REGION Network 4: 3号梯内呼指示灯绑定
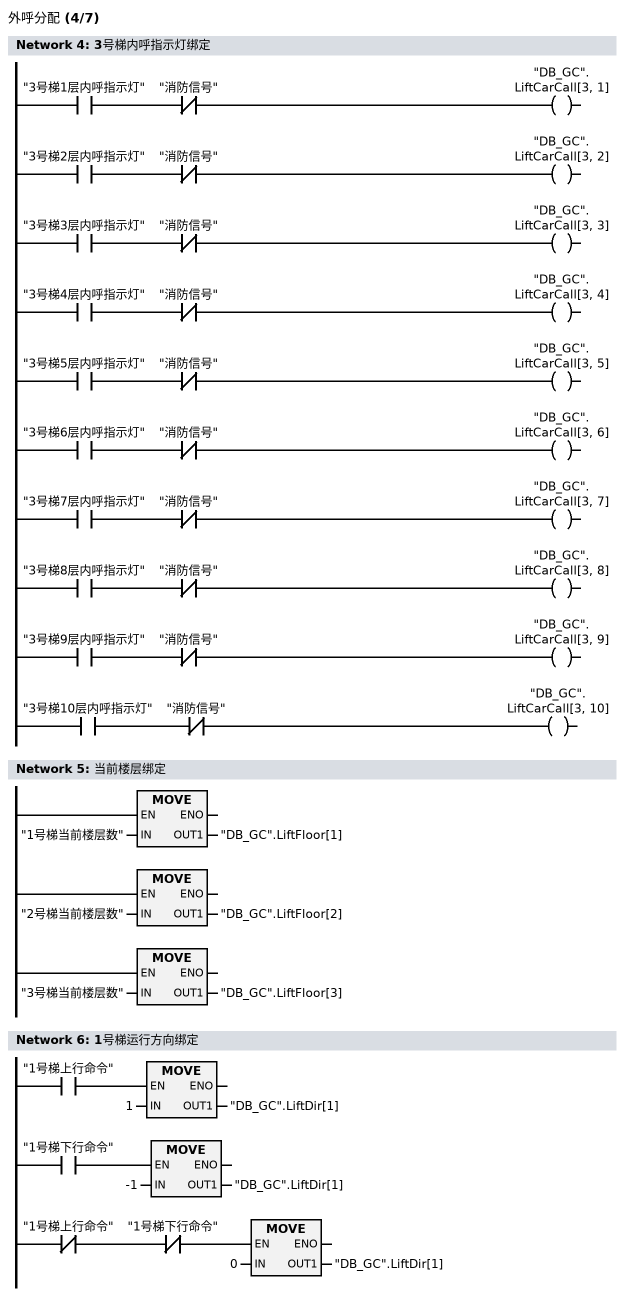
   RUNG wire#powerrail
      Contact( "3号梯1层内呼指示灯" )
      I_Contact( "消防信号" )
      Coil( "DB_GC".LiftCarCall[3, 1] )
   END_RUNG
   RUNG wire#powerrail
      Contact( "3号梯2层内呼指示灯" )
      I_Contact( "消防信号" )
      Coil( "DB_GC".LiftCarCall[3, 2] )
   END_RUNG
   RUNG wire#powerrail
      Contact( "3号梯3层内呼指示灯" )
      I_Contact( "消防信号" )
      Coil( "DB_GC".LiftCarCall[3, 3] )
   END_RUNG
   RUNG wire#powerrail
      Contact( "3号梯4层内呼指示灯" )
      I_Contact( "消防信号" )
      Coil( "DB_GC".LiftCarCall[3, 4] )
   END_RUNG
   RUNG wire#powerrail
      Contact( "3号梯5层内呼指示灯" )
      I_Contact( "消防信号" )
      Coil( "DB_GC".LiftCarCall[3, 5] )
   END_RUNG
   RUNG wire#powerrail
      Contact( "3号梯6层内呼指示灯" )
      I_Contact( "消防信号" )
      Coil( "DB_GC".LiftCarCall[3, 6] )
   END_RUNG
   RUNG wire#powerrail
      Contact( "3号梯7层内呼指示灯" )
      I_Contact( "消防信号" )
      Coil( "DB_GC".LiftCarCall[3, 7] )
   END_RUNG
   RUNG wire#powerrail
      Contact( "3号梯8层内呼指示灯" )
      I_Contact( "消防信号" )
      Coil( "DB_GC".LiftCarCall[3, 8] )
   END_RUNG
   RUNG wire#powerrail
      Contact( "3号梯9层内呼指示灯" )
      I_Contact( "消防信号" )
      Coil( "DB_GC".LiftCarCall[3, 9] )
   END_RUNG
   RUNG wire#powerrail
      Contact( "3号梯10层内呼指示灯" )
      I_Contact( "消防信号" )
      Coil( "DB_GC".LiftCarCall[3, 10] )
   END_RUNG
   // the same network as SCL:
   "DB_GC".LiftCarCall[3, 1] := "3号梯1层内呼指示灯" AND NOT "消防信号";
   "DB_GC".LiftCarCall[3, 2] := "3号梯2层内呼指示灯" AND NOT "消防信号";
   "DB_GC".LiftCarCall[3, 3] := "3号梯3层内呼指示灯" AND NOT "消防信号";
   "DB_GC".LiftCarCall[3, 4] := "3号梯4层内呼指示灯" AND NOT "消防信号";
   "DB_GC".LiftCarCall[3, 5] := "3号梯5层内呼指示灯" AND NOT "消防信号";
   "DB_GC".LiftCarCall[3, 6] := "3号梯6层内呼指示灯" AND NOT "消防信号";
   "DB_GC".LiftCarCall[3, 7] := "3号梯7层内呼指示灯" AND NOT "消防信号";
   "DB_GC".LiftCarCall[3, 8] := "3号梯8层内呼指示灯" AND NOT "消防信号";
   "DB_GC".LiftCarCall[3, 9] := "3号梯9层内呼指示灯" AND NOT "消防信号";
   "DB_GC".LiftCarCall[3, 10] := "3号梯10层内呼指示灯" AND NOT "消防信号";
END_REGION

REGION Network 5: 当前楼层绑定
   RUNG wire#powerrail
      Move(in := "1号梯当前楼层数", out1 => "DB_GC".LiftFloor[1])
   END_RUNG
   RUNG wire#powerrail
      Move(in := "2号梯当前楼层数", out1 => "DB_GC".LiftFloor[2])
   END_RUNG
   RUNG wire#powerrail
      Move(in := "3号梯当前楼层数", out1 => "DB_GC".LiftFloor[3])
   END_RUNG
   // the same network as SCL:
   "DB_GC".LiftFloor[1] := "1号梯当前楼层数";
   "DB_GC".LiftFloor[2] := "2号梯当前楼层数";
   "DB_GC".LiftFloor[3] := "3号梯当前楼层数";
END_REGION

REGION Network 6: 1号梯运行方向绑定
   RUNG wire#powerrail
      Contact( "1号梯上行命令" )
      Move(in := 1, out1 => "DB_GC".LiftDir[1])
   END_RUNG
   RUNG wire#powerrail
      Contact( "1号梯下行命令" )
      Move(in := -1, out1 => "DB_GC".LiftDir[1])
   END_RUNG
   RUNG wire#powerrail
      I_Contact( "1号梯上行命令" )
      I_Contact( "1号梯下行命令" )
      Move(in := 0, out1 => "DB_GC".LiftDir[1])
   END_RUNG
   // the same network as SCL:
   IF "1号梯上行命令" THEN "DB_GC".LiftDir[1] := 1; END_IF;
   IF "1号梯下行命令" THEN "DB_GC".LiftDir[1] := -1; END_IF;
   IF NOT "1号梯上行命令" AND NOT "1号梯下行命令" THEN "DB_GC".LiftDir[1] := 0; END_IF;
END_REGION

REGION Network 7: 2号梯运行方向绑定
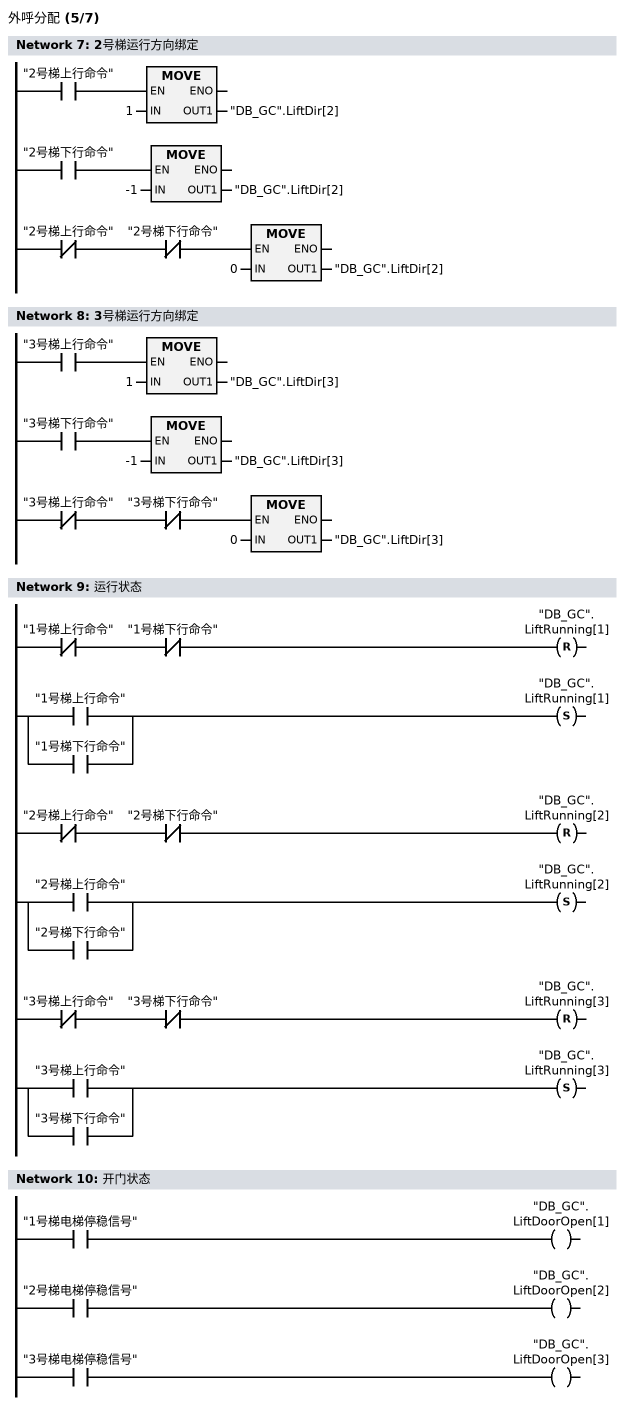
   RUNG wire#powerrail
      Contact( "2号梯上行命令" )
      Move(in := 1, out1 => "DB_GC".LiftDir[2])
   END_RUNG
   RUNG wire#powerrail
      Contact( "2号梯下行命令" )
      Move(in := -1, out1 => "DB_GC".LiftDir[2])
   END_RUNG
   RUNG wire#powerrail
      I_Contact( "2号梯上行命令" )
      I_Contact( "2号梯下行命令" )
      Move(in := 0, out1 => "DB_GC".LiftDir[2])
   END_RUNG
   // the same network as SCL:
   IF "2号梯上行命令" THEN "DB_GC".LiftDir[2] := 1; END_IF;
   IF "2号梯下行命令" THEN "DB_GC".LiftDir[2] := -1; END_IF;
   IF NOT "2号梯上行命令" AND NOT "2号梯下行命令" THEN "DB_GC".LiftDir[2] := 0; END_IF;
END_REGION

REGION Network 8: 3号梯运行方向绑定
   RUNG wire#powerrail
      Contact( "3号梯上行命令" )
      Move(in := 1, out1 => "DB_GC".LiftDir[3])
   END_RUNG
   RUNG wire#powerrail
      Contact( "3号梯下行命令" )
      Move(in := -1, out1 => "DB_GC".LiftDir[3])
   END_RUNG
   RUNG wire#powerrail
      I_Contact( "3号梯上行命令" )
      I_Contact( "3号梯下行命令" )
      Move(in := 0, out1 => "DB_GC".LiftDir[3])
   END_RUNG
   // the same network as SCL:
   IF "3号梯上行命令" THEN "DB_GC".LiftDir[3] := 1; END_IF;
   IF "3号梯下行命令" THEN "DB_GC".LiftDir[3] := -1; END_IF;
   IF NOT "3号梯上行命令" AND NOT "3号梯下行命令" THEN "DB_GC".LiftDir[3] := 0; END_IF;
END_REGION

REGION Network 9: 运行状态
   RUNG wire#powerrail
      I_Contact( "1号梯上行命令" )
      I_Contact( "1号梯下行命令" )
      R_Coil( "DB_GC".LiftRunning[1] )
   END_RUNG
   RUNG wire#powerrail
      Contact( "1号梯上行命令" )
      wire#w1
      S_Coil( "DB_GC".LiftRunning[1] )
   END_RUNG
   RUNG wire#powerrail
      Contact( "1号梯下行命令" )
   END_RUNG wire#w1
   RUNG wire#powerrail
      I_Contact( "2号梯上行命令" )
      I_Contact( "2号梯下行命令" )
      R_Coil( "DB_GC".LiftRunning[2] )
   END_RUNG
   RUNG wire#powerrail
      Contact( "2号梯上行命令" )
      wire#w2
      S_Coil( "DB_GC".LiftRunning[2] )
   END_RUNG
   RUNG wire#powerrail
      Contact( "2号梯下行命令" )
   END_RUNG wire#w2
   RUNG wire#powerrail
      I_Contact( "3号梯上行命令" )
      I_Contact( "3号梯下行命令" )
      R_Coil( "DB_GC".LiftRunning[3] )
   END_RUNG
   RUNG wire#powerrail
      Contact( "3号梯上行命令" )
      wire#w3
      S_Coil( "DB_GC".LiftRunning[3] )
   END_RUNG
   RUNG wire#powerrail
      Contact( "3号梯下行命令" )
   END_RUNG wire#w3
   // the same network as SCL:
   IF NOT "1号梯上行命令" AND NOT "1号梯下行命令" THEN "DB_GC".LiftRunning[1] := FALSE; END_IF;
   IF "1号梯上行命令" OR "1号梯下行命令" THEN "DB_GC".LiftRunning[1] := TRUE; END_IF;
   IF NOT "2号梯上行命令" AND NOT "2号梯下行命令" THEN "DB_GC".LiftRunning[2] := FALSE; END_IF;
   IF "2号梯上行命令" OR "2号梯下行命令" THEN "DB_GC".LiftRunning[2] := TRUE; END_IF;
   IF NOT "3号梯上行命令" AND NOT "3号梯下行命令" THEN "DB_GC".LiftRunning[3] := FALSE; END_IF;
   IF "3号梯上行命令" OR "3号梯下行命令" THEN "DB_GC".LiftRunning[3] := TRUE; END_IF;
END_REGION

REGION Network 10: 开门状态
   RUNG wire#powerrail
      Contact( "1号梯电梯停稳信号" )
      Coil( "DB_GC".LiftDoorOpen[1] )
   END_RUNG
   RUNG wire#powerrail
      Contact( "2号梯电梯停稳信号" )
      Coil( "DB_GC".LiftDoorOpen[2] )
   END_RUNG
   RUNG wire#powerrail
      Contact( "3号梯电梯停稳信号" )
      Coil( "DB_GC".LiftDoorOpen[3] )
   END_RUNG
   // the same network as SCL:
   "DB_GC".LiftDoorOpen[1] := "1号梯电梯停稳信号";
   "DB_GC".LiftDoorOpen[2] := "2号梯电梯停稳信号";
   "DB_GC".LiftDoorOpen[3] := "3号梯电梯停稳信号";
END_REGION

REGION Network 11: 锁梯
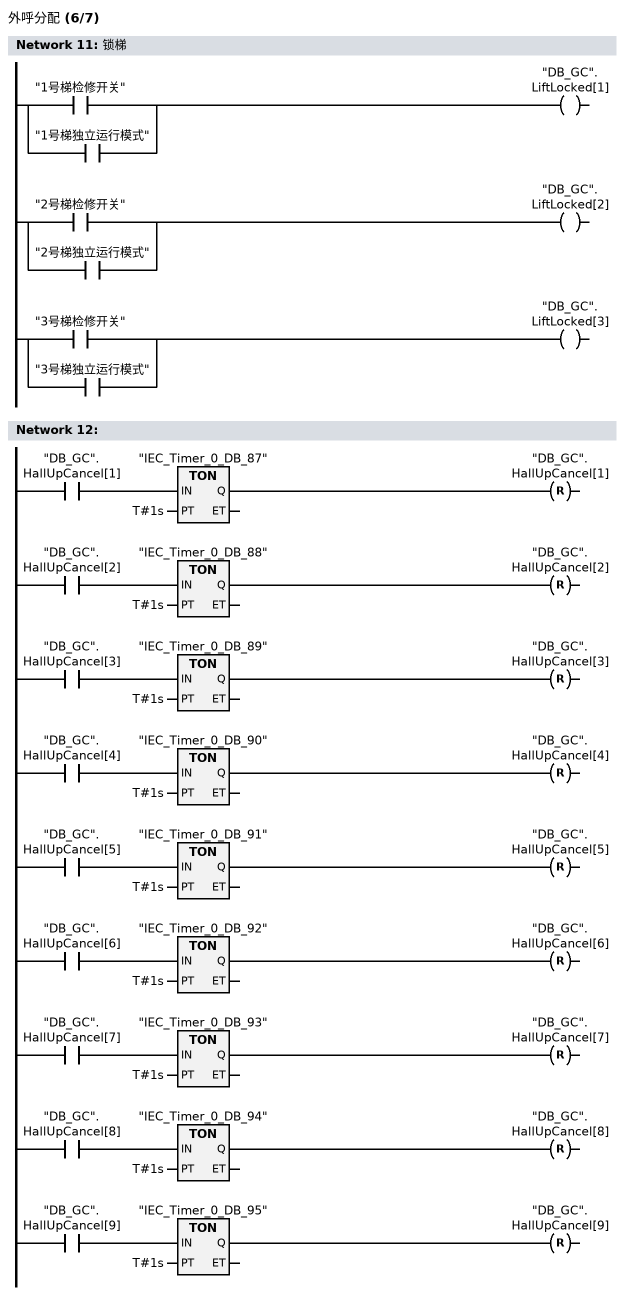
   RUNG wire#powerrail
      Contact( "1号梯检修开关" )
      wire#w1
      Coil( "DB_GC".LiftLocked[1] )
   END_RUNG
   RUNG wire#powerrail
      Contact( "1号梯独立运行模式" )
   END_RUNG wire#w1
   RUNG wire#powerrail
      Contact( "2号梯检修开关" )
      wire#w2
      Coil( "DB_GC".LiftLocked[2] )
   END_RUNG
   RUNG wire#powerrail
      Contact( "2号梯独立运行模式" )
   END_RUNG wire#w2
   RUNG wire#powerrail
      Contact( "3号梯检修开关" )
      wire#w3
      Coil( "DB_GC".LiftLocked[3] )
   END_RUNG
   RUNG wire#powerrail
      Contact( "3号梯独立运行模式" )
   END_RUNG wire#w3
   // the same network as SCL:
   "DB_GC".LiftLocked[1] := "1号梯检修开关" OR "1号梯独立运行模式";
   "DB_GC".LiftLocked[2] := "2号梯检修开关" OR "2号梯独立运行模式";
   "DB_GC".LiftLocked[3] := "3号梯检修开关" OR "3号梯独立运行模式";
END_REGION

REGION Network 12
   "IEC_Timer_0_DB_87".TON(IN := "DB_GC".HallUpCancel[1], PT := T#1s);
   IF "IEC_Timer_0_DB_87".Q THEN "DB_GC".HallUpCancel[1] := FALSE; END_IF;
   "IEC_Timer_0_DB_88".TON(IN := "DB_GC".HallUpCancel[2], PT := T#1s);
   IF "IEC_Timer_0_DB_88".Q THEN "DB_GC".HallUpCancel[2] := FALSE; END_IF;
   "IEC_Timer_0_DB_89".TON(IN := "DB_GC".HallUpCancel[3], PT := T#1s);
   IF "IEC_Timer_0_DB_89".Q THEN "DB_GC".HallUpCancel[3] := FALSE; END_IF;
   "IEC_Timer_0_DB_90".TON(IN := "DB_GC".HallUpCancel[4], PT := T#1s);
   IF "IEC_Timer_0_DB_90".Q THEN "DB_GC".HallUpCancel[4] := FALSE; END_IF;
   "IEC_Timer_0_DB_91".TON(IN := "DB_GC".HallUpCancel[5], PT := T#1s);
   IF "IEC_Timer_0_DB_91".Q THEN "DB_GC".HallUpCancel[5] := FALSE; END_IF;
   "IEC_Timer_0_DB_92".TON(IN := "DB_GC".HallUpCancel[6], PT := T#1s);
   IF "IEC_Timer_0_DB_92".Q THEN "DB_GC".HallUpCancel[6] := FALSE; END_IF;
   "IEC_Timer_0_DB_93".TON(IN := "DB_GC".HallUpCancel[7], PT := T#1s);
   IF "IEC_Timer_0_DB_93".Q THEN "DB_GC".HallUpCancel[7] := FALSE; END_IF;
   "IEC_Timer_0_DB_94".TON(IN := "DB_GC".HallUpCancel[8], PT := T#1s);
   IF "IEC_Timer_0_DB_94".Q THEN "DB_GC".HallUpCancel[8] := FALSE; END_IF;
   "IEC_Timer_0_DB_95".TON(IN := "DB_GC".HallUpCancel[9], PT := T#1s);
   IF "IEC_Timer_0_DB_95".Q THEN "DB_GC".HallUpCancel[9] := FALSE; END_IF;
END_REGION

REGION Network 13
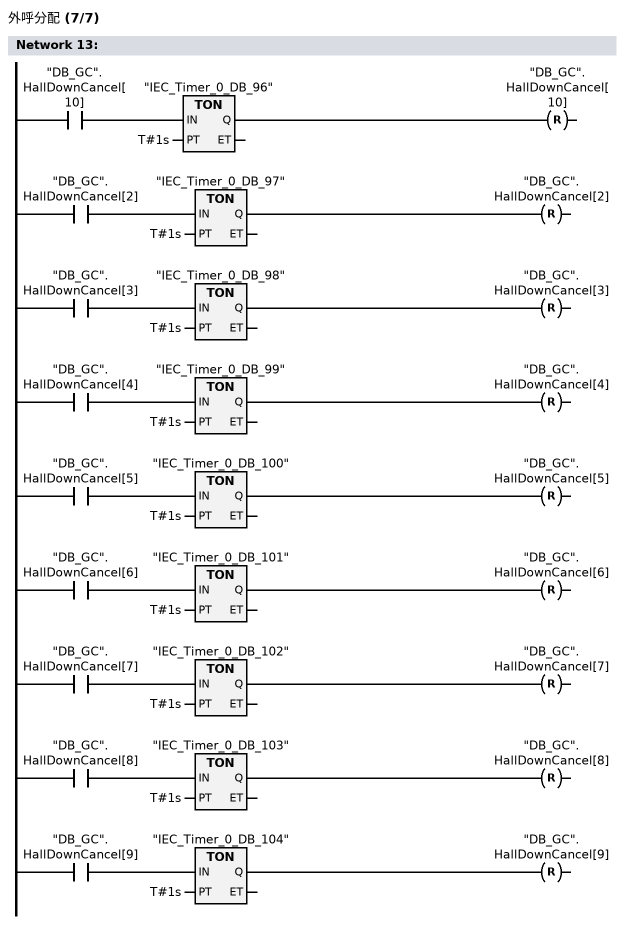
   "IEC_Timer_0_DB_96".TON(IN := "DB_GC".HallDownCancel[10], PT := T#1s);
   IF "IEC_Timer_0_DB_96".Q THEN "DB_GC".HallDownCancel[10] := FALSE; END_IF;
   "IEC_Timer_0_DB_97".TON(IN := "DB_GC".HallDownCancel[2], PT := T#1s);
   IF "IEC_Timer_0_DB_97".Q THEN "DB_GC".HallDownCancel[2] := FALSE; END_IF;
   "IEC_Timer_0_DB_98".TON(IN := "DB_GC".HallDownCancel[3], PT := T#1s);
   IF "IEC_Timer_0_DB_98".Q THEN "DB_GC".HallDownCancel[3] := FALSE; END_IF;
   "IEC_Timer_0_DB_99".TON(IN := "DB_GC".HallDownCancel[4], PT := T#1s);
   IF "IEC_Timer_0_DB_99".Q THEN "DB_GC".HallDownCancel[4] := FALSE; END_IF;
   "IEC_Timer_0_DB_100".TON(IN := "DB_GC".HallDownCancel[5], PT := T#1s);
   IF "IEC_Timer_0_DB_100".Q THEN "DB_GC".HallDownCancel[5] := FALSE; END_IF;
   "IEC_Timer_0_DB_101".TON(IN := "DB_GC".HallDownCancel[6], PT := T#1s);
   IF "IEC_Timer_0_DB_101".Q THEN "DB_GC".HallDownCancel[6] := FALSE; END_IF;
   "IEC_Timer_0_DB_102".TON(IN := "DB_GC".HallDownCancel[7], PT := T#1s);
   IF "IEC_Timer_0_DB_102".Q THEN "DB_GC".HallDownCancel[7] := FALSE; END_IF;
   "IEC_Timer_0_DB_103".TON(IN := "DB_GC".HallDownCancel[8], PT := T#1s);
   IF "IEC_Timer_0_DB_103".Q THEN "DB_GC".HallDownCancel[8] := FALSE; END_IF;
   "IEC_Timer_0_DB_104".TON(IN := "DB_GC".HallDownCancel[9], PT := T#1s);
   IF "IEC_Timer_0_DB_104".Q THEN "DB_GC".HallDownCancel[9] := FALSE; END_IF;
END_REGION
END_FUNCTION

FUNCTION "变量输出赋值" : Void   // FC2, LAD
{ S7_Optimized_Access := 'TRUE' }
VERSION : 0.1
   VAR_TEMP
      沿 : Bool;
   END_VAR
   VAR_TEMP   // added for the SCL form of the ladder/FBD networks
      _w1 : Bool;
   END_VAR
BEGIN

REGION Network 1: 1号梯内呼指示灯
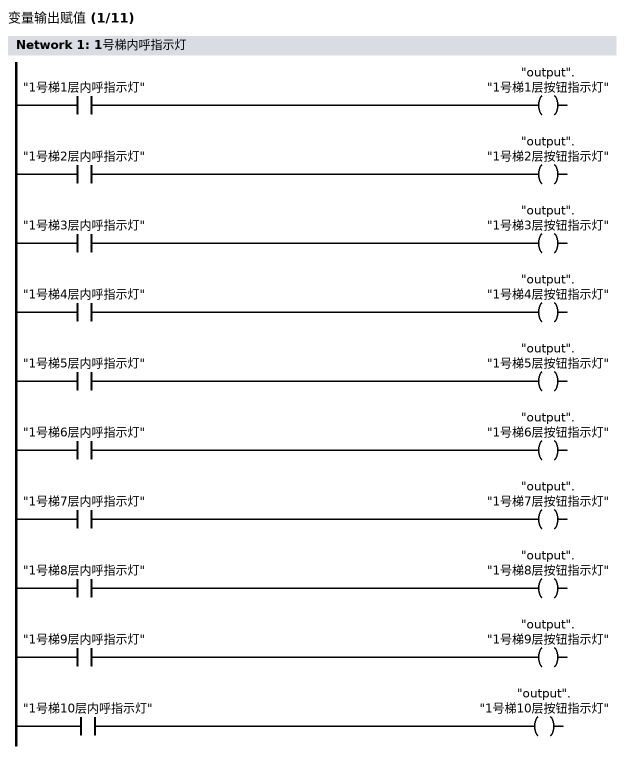
   RUNG wire#powerrail
      Contact( "1号梯1层内呼指示灯" )
      Coil( "output"."1号梯1层按钮指示灯" )
   END_RUNG
   RUNG wire#powerrail
      Contact( "1号梯2层内呼指示灯" )
      Coil( "output"."1号梯2层按钮指示灯" )
   END_RUNG
   RUNG wire#powerrail
      Contact( "1号梯3层内呼指示灯" )
      Coil( "output"."1号梯3层按钮指示灯" )
   END_RUNG
   RUNG wire#powerrail
      Contact( "1号梯4层内呼指示灯" )
      Coil( "output"."1号梯4层按钮指示灯" )
   END_RUNG
   RUNG wire#powerrail
      Contact( "1号梯5层内呼指示灯" )
      Coil( "output"."1号梯5层按钮指示灯" )
   END_RUNG
   RUNG wire#powerrail
      Contact( "1号梯6层内呼指示灯" )
      Coil( "output"."1号梯6层按钮指示灯" )
   END_RUNG
   RUNG wire#powerrail
      Contact( "1号梯7层内呼指示灯" )
      Coil( "output"."1号梯7层按钮指示灯" )
   END_RUNG
   RUNG wire#powerrail
      Contact( "1号梯8层内呼指示灯" )
      Coil( "output"."1号梯8层按钮指示灯" )
   END_RUNG
   RUNG wire#powerrail
      Contact( "1号梯9层内呼指示灯" )
      Coil( "output"."1号梯9层按钮指示灯" )
   END_RUNG
   RUNG wire#powerrail
      Contact( "1号梯10层内呼指示灯" )
      Coil( "output"."1号梯10层按钮指示灯" )
   END_RUNG
   // the same network as SCL:
   "output"."1号梯1层按钮指示灯" := "1号梯1层内呼指示灯";
   "output"."1号梯2层按钮指示灯" := "1号梯2层内呼指示灯";
   "output"."1号梯3层按钮指示灯" := "1号梯3层内呼指示灯";
   "output"."1号梯4层按钮指示灯" := "1号梯4层内呼指示灯";
   "output"."1号梯5层按钮指示灯" := "1号梯5层内呼指示灯";
   "output"."1号梯6层按钮指示灯" := "1号梯6层内呼指示灯";
   "output"."1号梯7层按钮指示灯" := "1号梯7层内呼指示灯";
   "output"."1号梯8层按钮指示灯" := "1号梯8层内呼指示灯";
   "output"."1号梯9层按钮指示灯" := "1号梯9层内呼指示灯";
   "output"."1号梯10层按钮指示灯" := "1号梯10层内呼指示灯";
END_REGION

REGION Network 2: 2号梯内呼指示灯
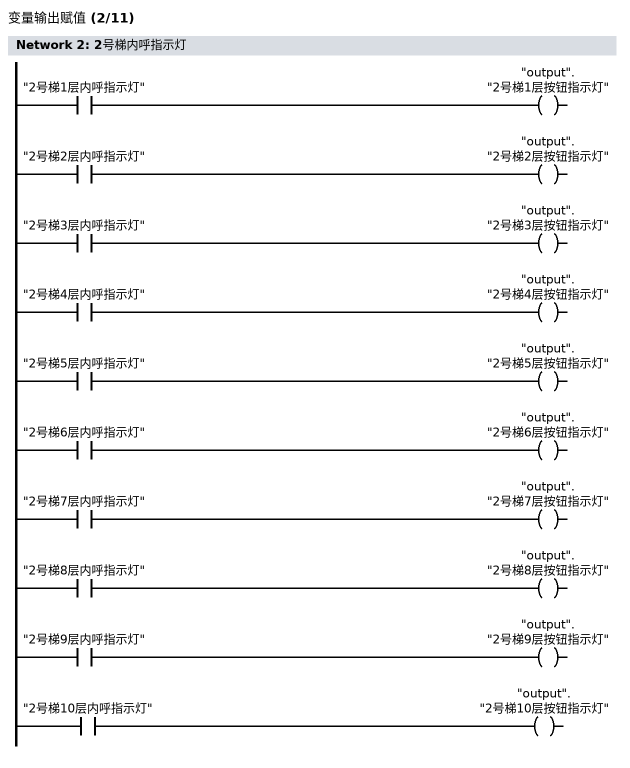
   RUNG wire#powerrail
      Contact( "2号梯1层内呼指示灯" )
      Coil( "output"."2号梯1层按钮指示灯" )
   END_RUNG
   RUNG wire#powerrail
      Contact( "2号梯2层内呼指示灯" )
      Coil( "output"."2号梯2层按钮指示灯" )
   END_RUNG
   RUNG wire#powerrail
      Contact( "2号梯3层内呼指示灯" )
      Coil( "output"."2号梯3层按钮指示灯" )
   END_RUNG
   RUNG wire#powerrail
      Contact( "2号梯4层内呼指示灯" )
      Coil( "output"."2号梯4层按钮指示灯" )
   END_RUNG
   RUNG wire#powerrail
      Contact( "2号梯5层内呼指示灯" )
      Coil( "output"."2号梯5层按钮指示灯" )
   END_RUNG
   RUNG wire#powerrail
      Contact( "2号梯6层内呼指示灯" )
      Coil( "output"."2号梯6层按钮指示灯" )
   END_RUNG
   RUNG wire#powerrail
      Contact( "2号梯7层内呼指示灯" )
      Coil( "output"."2号梯7层按钮指示灯" )
   END_RUNG
   RUNG wire#powerrail
      Contact( "2号梯8层内呼指示灯" )
      Coil( "output"."2号梯8层按钮指示灯" )
   END_RUNG
   RUNG wire#powerrail
      Contact( "2号梯9层内呼指示灯" )
      Coil( "output"."2号梯9层按钮指示灯" )
   END_RUNG
   RUNG wire#powerrail
      Contact( "2号梯10层内呼指示灯" )
      Coil( "output"."2号梯10层按钮指示灯" )
   END_RUNG
   // the same network as SCL:
   "output"."2号梯1层按钮指示灯" := "2号梯1层内呼指示灯";
   "output"."2号梯2层按钮指示灯" := "2号梯2层内呼指示灯";
   "output"."2号梯3层按钮指示灯" := "2号梯3层内呼指示灯";
   "output"."2号梯4层按钮指示灯" := "2号梯4层内呼指示灯";
   "output"."2号梯5层按钮指示灯" := "2号梯5层内呼指示灯";
   "output"."2号梯6层按钮指示灯" := "2号梯6层内呼指示灯";
   "output"."2号梯7层按钮指示灯" := "2号梯7层内呼指示灯";
   "output"."2号梯8层按钮指示灯" := "2号梯8层内呼指示灯";
   "output"."2号梯9层按钮指示灯" := "2号梯9层内呼指示灯";
   "output"."2号梯10层按钮指示灯" := "2号梯10层内呼指示灯";
END_REGION

REGION Network 3: 3号梯内呼指示灯
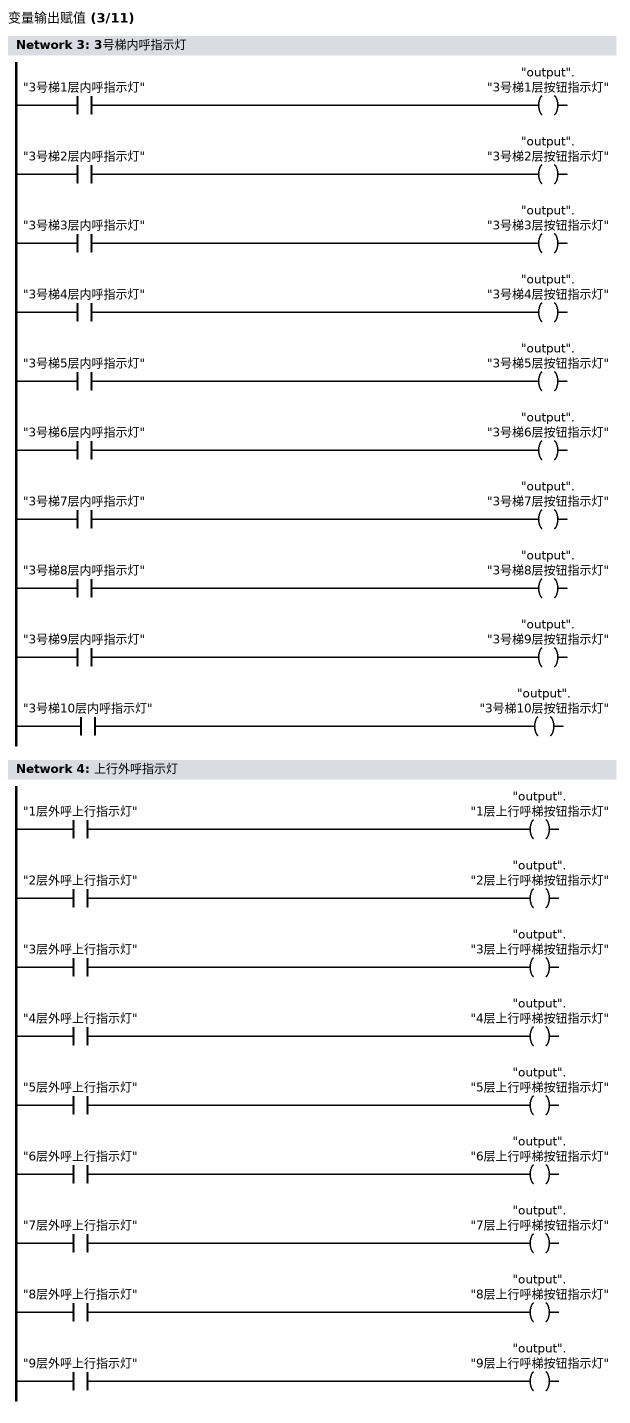
   RUNG wire#powerrail
      Contact( "3号梯1层内呼指示灯" )
      Coil( "output"."3号梯1层按钮指示灯" )
   END_RUNG
   RUNG wire#powerrail
      Contact( "3号梯2层内呼指示灯" )
      Coil( "output"."3号梯2层按钮指示灯" )
   END_RUNG
   RUNG wire#powerrail
      Contact( "3号梯3层内呼指示灯" )
      Coil( "output"."3号梯3层按钮指示灯" )
   END_RUNG
   RUNG wire#powerrail
      Contact( "3号梯4层内呼指示灯" )
      Coil( "output"."3号梯4层按钮指示灯" )
   END_RUNG
   RUNG wire#powerrail
      Contact( "3号梯5层内呼指示灯" )
      Coil( "output"."3号梯5层按钮指示灯" )
   END_RUNG
   RUNG wire#powerrail
      Contact( "3号梯6层内呼指示灯" )
      Coil( "output"."3号梯6层按钮指示灯" )
   END_RUNG
   RUNG wire#powerrail
      Contact( "3号梯7层内呼指示灯" )
      Coil( "output"."3号梯7层按钮指示灯" )
   END_RUNG
   RUNG wire#powerrail
      Contact( "3号梯8层内呼指示灯" )
      Coil( "output"."3号梯8层按钮指示灯" )
   END_RUNG
   RUNG wire#powerrail
      Contact( "3号梯9层内呼指示灯" )
      Coil( "output"."3号梯9层按钮指示灯" )
   END_RUNG
   RUNG wire#powerrail
      Contact( "3号梯10层内呼指示灯" )
      Coil( "output"."3号梯10层按钮指示灯" )
   END_RUNG
   // the same network as SCL:
   "output"."3号梯1层按钮指示灯" := "3号梯1层内呼指示灯";
   "output"."3号梯2层按钮指示灯" := "3号梯2层内呼指示灯";
   "output"."3号梯3层按钮指示灯" := "3号梯3层内呼指示灯";
   "output"."3号梯4层按钮指示灯" := "3号梯4层内呼指示灯";
   "output"."3号梯5层按钮指示灯" := "3号梯5层内呼指示灯";
   "output"."3号梯6层按钮指示灯" := "3号梯6层内呼指示灯";
   "output"."3号梯7层按钮指示灯" := "3号梯7层内呼指示灯";
   "output"."3号梯8层按钮指示灯" := "3号梯8层内呼指示灯";
   "output"."3号梯9层按钮指示灯" := "3号梯9层内呼指示灯";
   "output"."3号梯10层按钮指示灯" := "3号梯10层内呼指示灯";
END_REGION

REGION Network 4: 上行外呼指示灯
   RUNG wire#powerrail
      Contact( "1层外呼上行指示灯" )
      Coil( "output"."1层上行呼梯按钮指示灯" )
   END_RUNG
   RUNG wire#powerrail
      Contact( "2层外呼上行指示灯" )
      Coil( "output"."2层上行呼梯按钮指示灯" )
   END_RUNG
   RUNG wire#powerrail
      Contact( "3层外呼上行指示灯" )
      Coil( "output"."3层上行呼梯按钮指示灯" )
   END_RUNG
   RUNG wire#powerrail
      Contact( "4层外呼上行指示灯" )
      Coil( "output"."4层上行呼梯按钮指示灯" )
   END_RUNG
   RUNG wire#powerrail
      Contact( "5层外呼上行指示灯" )
      Coil( "output"."5层上行呼梯按钮指示灯" )
   END_RUNG
   RUNG wire#powerrail
      Contact( "6层外呼上行指示灯" )
      Coil( "output"."6层上行呼梯按钮指示灯" )
   END_RUNG
   RUNG wire#powerrail
      Contact( "7层外呼上行指示灯" )
      Coil( "output"."7层上行呼梯按钮指示灯" )
   END_RUNG
   RUNG wire#powerrail
      Contact( "8层外呼上行指示灯" )
      Coil( "output"."8层上行呼梯按钮指示灯" )
   END_RUNG
   RUNG wire#powerrail
      Contact( "9层外呼上行指示灯" )
      Coil( "output"."9层上行呼梯按钮指示灯" )
   END_RUNG
   // the same network as SCL:
   "output"."1层上行呼梯按钮指示灯" := "1层外呼上行指示灯";
   "output"."2层上行呼梯按钮指示灯" := "2层外呼上行指示灯";
   "output"."3层上行呼梯按钮指示灯" := "3层外呼上行指示灯";
   "output"."4层上行呼梯按钮指示灯" := "4层外呼上行指示灯";
   "output"."5层上行呼梯按钮指示灯" := "5层外呼上行指示灯";
   "output"."6层上行呼梯按钮指示灯" := "6层外呼上行指示灯";
   "output"."7层上行呼梯按钮指示灯" := "7层外呼上行指示灯";
   "output"."8层上行呼梯按钮指示灯" := "8层外呼上行指示灯";
   "output"."9层上行呼梯按钮指示灯" := "9层外呼上行指示灯";
END_REGION

REGION Network 5: 下行外呼指示灯
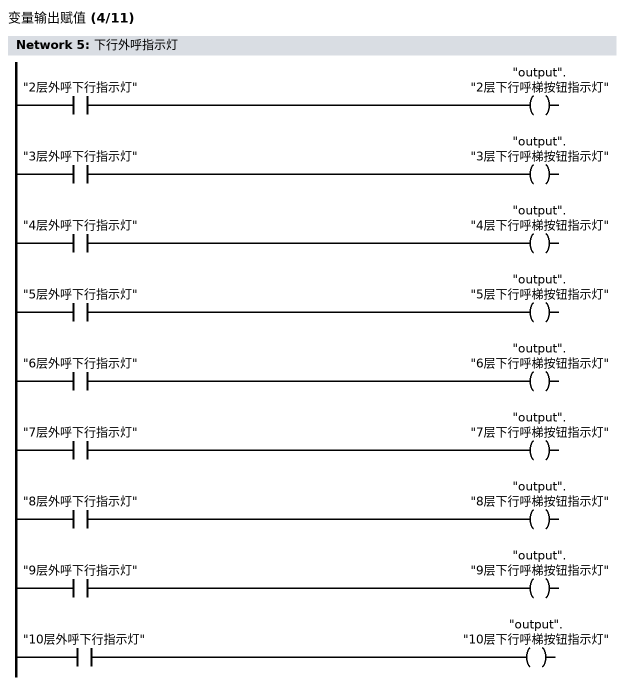
   RUNG wire#powerrail
      Contact( "2层外呼下行指示灯" )
      Coil( "output"."2层下行呼梯按钮指示灯" )
   END_RUNG
   RUNG wire#powerrail
      Contact( "3层外呼下行指示灯" )
      Coil( "output"."3层下行呼梯按钮指示灯" )
   END_RUNG
   RUNG wire#powerrail
      Contact( "4层外呼下行指示灯" )
      Coil( "output"."4层下行呼梯按钮指示灯" )
   END_RUNG
   RUNG wire#powerrail
      Contact( "5层外呼下行指示灯" )
      Coil( "output"."5层下行呼梯按钮指示灯" )
   END_RUNG
   RUNG wire#powerrail
      Contact( "6层外呼下行指示灯" )
      Coil( "output"."6层下行呼梯按钮指示灯" )
   END_RUNG
   RUNG wire#powerrail
      Contact( "7层外呼下行指示灯" )
      Coil( "output"."7层下行呼梯按钮指示灯" )
   END_RUNG
   RUNG wire#powerrail
      Contact( "8层外呼下行指示灯" )
      Coil( "output"."8层下行呼梯按钮指示灯" )
   END_RUNG
   RUNG wire#powerrail
      Contact( "9层外呼下行指示灯" )
      Coil( "output"."9层下行呼梯按钮指示灯" )
   END_RUNG
   RUNG wire#powerrail
      Contact( "10层外呼下行指示灯" )
      Coil( "output"."10层下行呼梯按钮指示灯" )
   END_RUNG
   // the same network as SCL:
   "output"."2层下行呼梯按钮指示灯" := "2层外呼下行指示灯";
   "output"."3层下行呼梯按钮指示灯" := "3层外呼下行指示灯";
   "output"."4层下行呼梯按钮指示灯" := "4层外呼下行指示灯";
   "output"."5层下行呼梯按钮指示灯" := "5层外呼下行指示灯";
   "output"."6层下行呼梯按钮指示灯" := "6层外呼下行指示灯";
   "output"."7层下行呼梯按钮指示灯" := "7层外呼下行指示灯";
   "output"."8层下行呼梯按钮指示灯" := "8层外呼下行指示灯";
   "output"."9层下行呼梯按钮指示灯" := "9层外呼下行指示灯";
   "output"."10层下行呼梯按钮指示灯" := "10层外呼下行指示灯";
END_REGION

REGION Network 6: 1号梯数码管显示
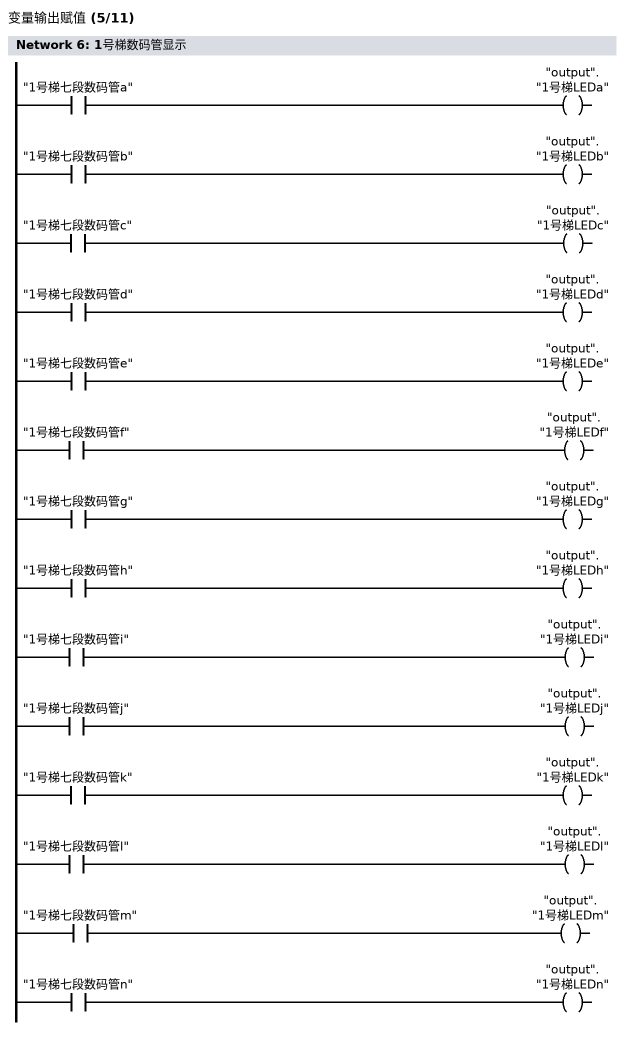
   RUNG wire#powerrail
      Contact( "1号梯七段数码管a" )
      Coil( "output"."1号梯LEDa" )
   END_RUNG
   RUNG wire#powerrail
      Contact( "1号梯七段数码管b" )
      Coil( "output"."1号梯LEDb" )
   END_RUNG
   RUNG wire#powerrail
      Contact( "1号梯七段数码管c" )
      Coil( "output"."1号梯LEDc" )
   END_RUNG
   RUNG wire#powerrail
      Contact( "1号梯七段数码管d" )
      Coil( "output"."1号梯LEDd" )
   END_RUNG
   RUNG wire#powerrail
      Contact( "1号梯七段数码管e" )
      Coil( "output"."1号梯LEDe" )
   END_RUNG
   RUNG wire#powerrail
      Contact( "1号梯七段数码管f" )
      Coil( "output"."1号梯LEDf" )
   END_RUNG
   RUNG wire#powerrail
      Contact( "1号梯七段数码管g" )
      Coil( "output"."1号梯LEDg" )
   END_RUNG
   RUNG wire#powerrail
      Contact( "1号梯七段数码管h" )
      Coil( "output"."1号梯LEDh" )
   END_RUNG
   RUNG wire#powerrail
      Contact( "1号梯七段数码管i" )
      Coil( "output"."1号梯LEDi" )
   END_RUNG
   RUNG wire#powerrail
      Contact( "1号梯七段数码管j" )
      Coil( "output"."1号梯LEDj" )
   END_RUNG
   RUNG wire#powerrail
      Contact( "1号梯七段数码管k" )
      Coil( "output"."1号梯LEDk" )
   END_RUNG
   RUNG wire#powerrail
      Contact( "1号梯七段数码管l" )
      Coil( "output"."1号梯LEDl" )
   END_RUNG
   RUNG wire#powerrail
      Contact( "1号梯七段数码管m" )
      Coil( "output"."1号梯LEDm" )
   END_RUNG
   RUNG wire#powerrail
      Contact( "1号梯七段数码管n" )
      Coil( "output"."1号梯LEDn" )
   END_RUNG
   // the same network as SCL:
   "output"."1号梯LEDa" := "1号梯七段数码管a";
   "output"."1号梯LEDb" := "1号梯七段数码管b";
   "output"."1号梯LEDc" := "1号梯七段数码管c";
   "output"."1号梯LEDd" := "1号梯七段数码管d";
   "output"."1号梯LEDe" := "1号梯七段数码管e";
   "output"."1号梯LEDf" := "1号梯七段数码管f";
   "output"."1号梯LEDg" := "1号梯七段数码管g";
   "output"."1号梯LEDh" := "1号梯七段数码管h";
   "output"."1号梯LEDi" := "1号梯七段数码管i";
   "output"."1号梯LEDj" := "1号梯七段数码管j";
   "output"."1号梯LEDk" := "1号梯七段数码管k";
   "output"."1号梯LEDl" := "1号梯七段数码管l";
   "output"."1号梯LEDm" := "1号梯七段数码管m";
   "output"."1号梯LEDn" := "1号梯七段数码管n";
END_REGION

REGION Network 7: 2号梯数码管显示
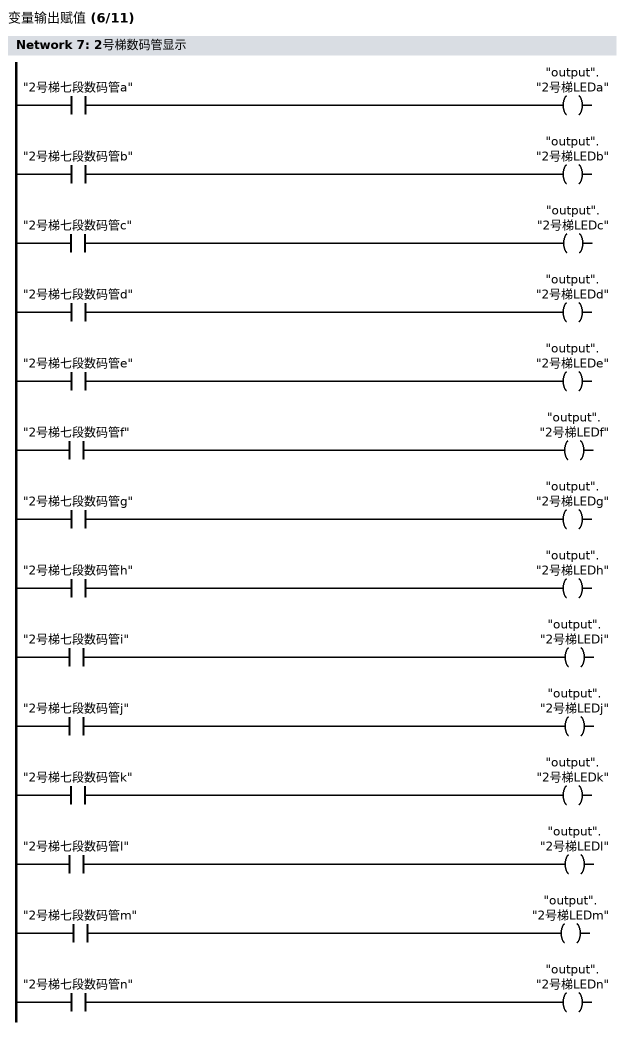
   RUNG wire#powerrail
      Contact( "2号梯七段数码管a" )
      Coil( "output"."2号梯LEDa" )
   END_RUNG
   RUNG wire#powerrail
      Contact( "2号梯七段数码管b" )
      Coil( "output"."2号梯LEDb" )
   END_RUNG
   RUNG wire#powerrail
      Contact( "2号梯七段数码管c" )
      Coil( "output"."2号梯LEDc" )
   END_RUNG
   RUNG wire#powerrail
      Contact( "2号梯七段数码管d" )
      Coil( "output"."2号梯LEDd" )
   END_RUNG
   RUNG wire#powerrail
      Contact( "2号梯七段数码管e" )
      Coil( "output"."2号梯LEDe" )
   END_RUNG
   RUNG wire#powerrail
      Contact( "2号梯七段数码管f" )
      Coil( "output"."2号梯LEDf" )
   END_RUNG
   RUNG wire#powerrail
      Contact( "2号梯七段数码管g" )
      Coil( "output"."2号梯LEDg" )
   END_RUNG
   RUNG wire#powerrail
      Contact( "2号梯七段数码管h" )
      Coil( "output"."2号梯LEDh" )
   END_RUNG
   RUNG wire#powerrail
      Contact( "2号梯七段数码管i" )
      Coil( "output"."2号梯LEDi" )
   END_RUNG
   RUNG wire#powerrail
      Contact( "2号梯七段数码管j" )
      Coil( "output"."2号梯LEDj" )
   END_RUNG
   RUNG wire#powerrail
      Contact( "2号梯七段数码管k" )
      Coil( "output"."2号梯LEDk" )
   END_RUNG
   RUNG wire#powerrail
      Contact( "2号梯七段数码管l" )
      Coil( "output"."2号梯LEDl" )
   END_RUNG
   RUNG wire#powerrail
      Contact( "2号梯七段数码管m" )
      Coil( "output"."2号梯LEDm" )
   END_RUNG
   RUNG wire#powerrail
      Contact( "2号梯七段数码管n" )
      Coil( "output"."2号梯LEDn" )
   END_RUNG
   // the same network as SCL:
   "output"."2号梯LEDa" := "2号梯七段数码管a";
   "output"."2号梯LEDb" := "2号梯七段数码管b";
   "output"."2号梯LEDc" := "2号梯七段数码管c";
   "output"."2号梯LEDd" := "2号梯七段数码管d";
   "output"."2号梯LEDe" := "2号梯七段数码管e";
   "output"."2号梯LEDf" := "2号梯七段数码管f";
   "output"."2号梯LEDg" := "2号梯七段数码管g";
   "output"."2号梯LEDh" := "2号梯七段数码管h";
   "output"."2号梯LEDi" := "2号梯七段数码管i";
   "output"."2号梯LEDj" := "2号梯七段数码管j";
   "output"."2号梯LEDk" := "2号梯七段数码管k";
   "output"."2号梯LEDl" := "2号梯七段数码管l";
   "output"."2号梯LEDm" := "2号梯七段数码管m";
   "output"."2号梯LEDn" := "2号梯七段数码管n";
END_REGION

REGION Network 8: 3号梯数码管显示
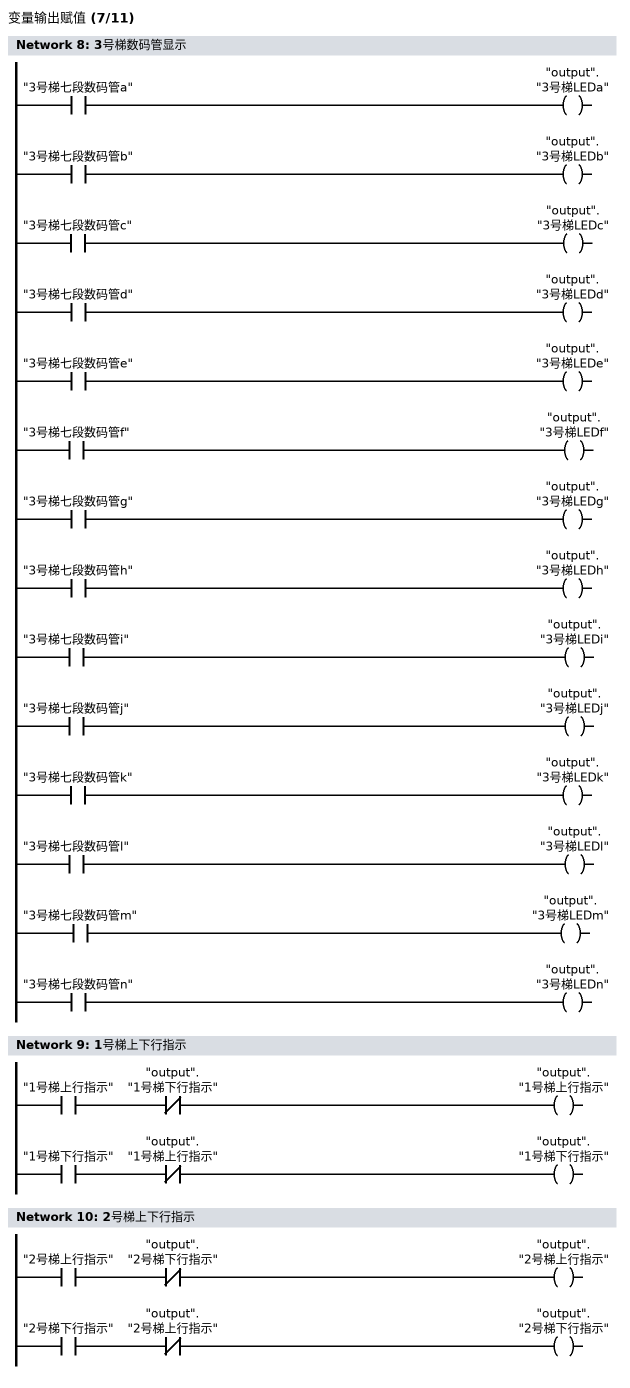
   RUNG wire#powerrail
      Contact( "3号梯七段数码管a" )
      Coil( "output"."3号梯LEDa" )
   END_RUNG
   RUNG wire#powerrail
      Contact( "3号梯七段数码管b" )
      Coil( "output"."3号梯LEDb" )
   END_RUNG
   RUNG wire#powerrail
      Contact( "3号梯七段数码管c" )
      Coil( "output"."3号梯LEDc" )
   END_RUNG
   RUNG wire#powerrail
      Contact( "3号梯七段数码管d" )
      Coil( "output"."3号梯LEDd" )
   END_RUNG
   RUNG wire#powerrail
      Contact( "3号梯七段数码管e" )
      Coil( "output"."3号梯LEDe" )
   END_RUNG
   RUNG wire#powerrail
      Contact( "3号梯七段数码管f" )
      Coil( "output"."3号梯LEDf" )
   END_RUNG
   RUNG wire#powerrail
      Contact( "3号梯七段数码管g" )
      Coil( "output"."3号梯LEDg" )
   END_RUNG
   RUNG wire#powerrail
      Contact( "3号梯七段数码管h" )
      Coil( "output"."3号梯LEDh" )
   END_RUNG
   RUNG wire#powerrail
      Contact( "3号梯七段数码管i" )
      Coil( "output"."3号梯LEDi" )
   END_RUNG
   RUNG wire#powerrail
      Contact( "3号梯七段数码管j" )
      Coil( "output"."3号梯LEDj" )
   END_RUNG
   RUNG wire#powerrail
      Contact( "3号梯七段数码管k" )
      Coil( "output"."3号梯LEDk" )
   END_RUNG
   RUNG wire#powerrail
      Contact( "3号梯七段数码管l" )
      Coil( "output"."3号梯LEDl" )
   END_RUNG
   RUNG wire#powerrail
      Contact( "3号梯七段数码管m" )
      Coil( "output"."3号梯LEDm" )
   END_RUNG
   RUNG wire#powerrail
      Contact( "3号梯七段数码管n" )
      Coil( "output"."3号梯LEDn" )
   END_RUNG
   // the same network as SCL:
   "output"."3号梯LEDa" := "3号梯七段数码管a";
   "output"."3号梯LEDb" := "3号梯七段数码管b";
   "output"."3号梯LEDc" := "3号梯七段数码管c";
   "output"."3号梯LEDd" := "3号梯七段数码管d";
   "output"."3号梯LEDe" := "3号梯七段数码管e";
   "output"."3号梯LEDf" := "3号梯七段数码管f";
   "output"."3号梯LEDg" := "3号梯七段数码管g";
   "output"."3号梯LEDh" := "3号梯七段数码管h";
   "output"."3号梯LEDi" := "3号梯七段数码管i";
   "output"."3号梯LEDj" := "3号梯七段数码管j";
   "output"."3号梯LEDk" := "3号梯七段数码管k";
   "output"."3号梯LEDl" := "3号梯七段数码管l";
   "output"."3号梯LEDm" := "3号梯七段数码管m";
   "output"."3号梯LEDn" := "3号梯七段数码管n";
END_REGION

REGION Network 9: 1号梯上下行指示
   RUNG wire#powerrail
      Contact( "1号梯上行指示" )
      I_Contact( "output"."1号梯下行指示" )
      Coil( "output"."1号梯上行指示" )
   END_RUNG
   RUNG wire#powerrail
      Contact( "1号梯下行指示" )
      I_Contact( "output"."1号梯上行指示" )
      Coil( "output"."1号梯下行指示" )
   END_RUNG
   // the same network as SCL:
   "output"."1号梯上行指示" := "1号梯上行指示" AND NOT "output"."1号梯下行指示";
   "output"."1号梯下行指示" := "1号梯下行指示" AND NOT "output"."1号梯上行指示";
END_REGION

REGION Network 10: 2号梯上下行指示
   RUNG wire#powerrail
      Contact( "2号梯上行指示" )
      I_Contact( "output"."2号梯下行指示" )
      Coil( "output"."2号梯上行指示" )
   END_RUNG
   RUNG wire#powerrail
      Contact( "2号梯下行指示" )
      I_Contact( "output"."2号梯上行指示" )
      Coil( "output"."2号梯下行指示" )
   END_RUNG
   // the same network as SCL:
   "output"."2号梯上行指示" := "2号梯上行指示" AND NOT "output"."2号梯下行指示";
   "output"."2号梯下行指示" := "2号梯下行指示" AND NOT "output"."2号梯上行指示";
END_REGION

REGION Network 11: 3号梯上下行指示
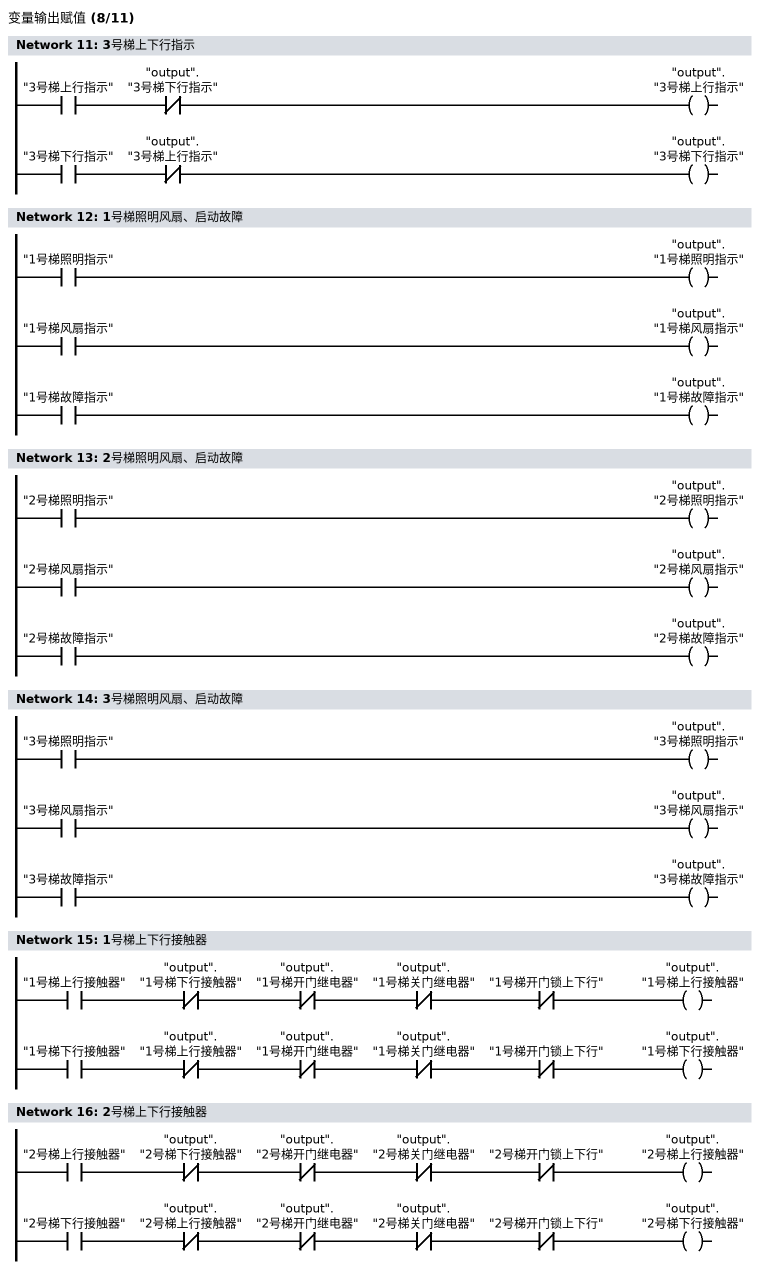
   RUNG wire#powerrail
      Contact( "3号梯上行指示" )
      I_Contact( "output"."3号梯下行指示" )
      Coil( "output"."3号梯上行指示" )
   END_RUNG
   RUNG wire#powerrail
      Contact( "3号梯下行指示" )
      I_Contact( "output"."3号梯上行指示" )
      Coil( "output"."3号梯下行指示" )
   END_RUNG
   // the same network as SCL:
   "output"."3号梯上行指示" := "3号梯上行指示" AND NOT "output"."3号梯下行指示";
   "output"."3号梯下行指示" := "3号梯下行指示" AND NOT "output"."3号梯上行指示";
END_REGION

REGION Network 12: 1号梯照明风扇、启动故障
   RUNG wire#powerrail
      Contact( "1号梯照明指示" )
      Coil( "output"."1号梯照明指示" )
   END_RUNG
   RUNG wire#powerrail
      Contact( "1号梯风扇指示" )
      Coil( "output"."1号梯风扇指示" )
   END_RUNG
   RUNG wire#powerrail
      Contact( "1号梯故障指示" )
      Coil( "output"."1号梯故障指示" )
   END_RUNG
   // the same network as SCL:
   "output"."1号梯照明指示" := "1号梯照明指示";
   "output"."1号梯风扇指示" := "1号梯风扇指示";
   "output"."1号梯故障指示" := "1号梯故障指示";
END_REGION

REGION Network 13: 2号梯照明风扇、启动故障
   RUNG wire#powerrail
      Contact( "2号梯照明指示" )
      Coil( "output"."2号梯照明指示" )
   END_RUNG
   RUNG wire#powerrail
      Contact( "2号梯风扇指示" )
      Coil( "output"."2号梯风扇指示" )
   END_RUNG
   RUNG wire#powerrail
      Contact( "2号梯故障指示" )
      Coil( "output"."2号梯故障指示" )
   END_RUNG
   // the same network as SCL:
   "output"."2号梯照明指示" := "2号梯照明指示";
   "output"."2号梯风扇指示" := "2号梯风扇指示";
   "output"."2号梯故障指示" := "2号梯故障指示";
END_REGION

REGION Network 14: 3号梯照明风扇、启动故障
   RUNG wire#powerrail
      Contact( "3号梯照明指示" )
      Coil( "output"."3号梯照明指示" )
   END_RUNG
   RUNG wire#powerrail
      Contact( "3号梯风扇指示" )
      Coil( "output"."3号梯风扇指示" )
   END_RUNG
   RUNG wire#powerrail
      Contact( "3号梯故障指示" )
      Coil( "output"."3号梯故障指示" )
   END_RUNG
   // the same network as SCL:
   "output"."3号梯照明指示" := "3号梯照明指示";
   "output"."3号梯风扇指示" := "3号梯风扇指示";
   "output"."3号梯故障指示" := "3号梯故障指示";
END_REGION

REGION Network 15: 1号梯上下行接触器
   RUNG wire#powerrail
      Contact( "1号梯上行接触器" )
      I_Contact( "output"."1号梯下行接触器" )
      I_Contact( "output"."1号梯开门继电器" )
      I_Contact( "output"."1号梯关门继电器" )
      I_Contact( "1号梯开门锁上下行" )
      Coil( "output"."1号梯上行接触器" )
   END_RUNG
   RUNG wire#powerrail
      Contact( "1号梯下行接触器" )
      I_Contact( "output"."1号梯上行接触器" )
      I_Contact( "output"."1号梯开门继电器" )
      I_Contact( "output"."1号梯关门继电器" )
      I_Contact( "1号梯开门锁上下行" )
      Coil( "output"."1号梯下行接触器" )
   END_RUNG
   // the same network as SCL:
   "output"."1号梯上行接触器" := "1号梯上行接触器" AND NOT "output"."1号梯下行接触器" AND NOT "output"."1号梯开门继电器" AND NOT "output"."1号梯关门继电器" AND NOT "1号梯开门锁上下行";
   "output"."1号梯下行接触器" := "1号梯下行接触器" AND NOT "output"."1号梯上行接触器" AND NOT "output"."1号梯开门继电器" AND NOT "output"."1号梯关门继电器" AND NOT "1号梯开门锁上下行";
END_REGION

REGION Network 16: 2号梯上下行接触器
   RUNG wire#powerrail
      Contact( "2号梯上行接触器" )
      I_Contact( "output"."2号梯下行接触器" )
      I_Contact( "output"."2号梯开门继电器" )
      I_Contact( "output"."2号梯关门继电器" )
      I_Contact( "2号梯开门锁上下行" )
      Coil( "output"."2号梯上行接触器" )
   END_RUNG
   RUNG wire#powerrail
      Contact( "2号梯下行接触器" )
      I_Contact( "output"."2号梯上行接触器" )
      I_Contact( "output"."2号梯开门继电器" )
      I_Contact( "output"."2号梯关门继电器" )
      I_Contact( "2号梯开门锁上下行" )
      Coil( "output"."2号梯下行接触器" )
   END_RUNG
   // the same network as SCL:
   "output"."2号梯上行接触器" := "2号梯上行接触器" AND NOT "output"."2号梯下行接触器" AND NOT "output"."2号梯开门继电器" AND NOT "output"."2号梯关门继电器" AND NOT "2号梯开门锁上下行";
   "output"."2号梯下行接触器" := "2号梯下行接触器" AND NOT "output"."2号梯上行接触器" AND NOT "output"."2号梯开门继电器" AND NOT "output"."2号梯关门继电器" AND NOT "2号梯开门锁上下行";
END_REGION

REGION Network 17: 3号梯上下行接触器
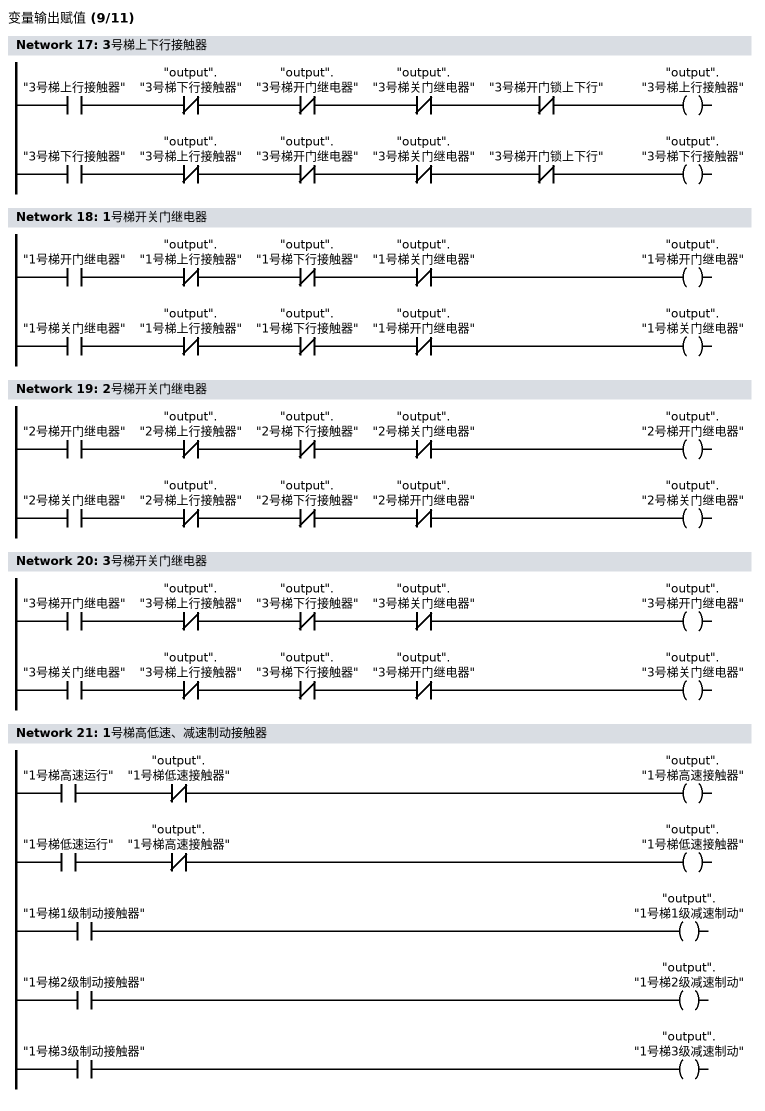
   RUNG wire#powerrail
      Contact( "3号梯上行接触器" )
      I_Contact( "output"."3号梯下行接触器" )
      I_Contact( "output"."3号梯开门继电器" )
      I_Contact( "output"."3号梯关门继电器" )
      I_Contact( "3号梯开门锁上下行" )
      Coil( "output"."3号梯上行接触器" )
   END_RUNG
   RUNG wire#powerrail
      Contact( "3号梯下行接触器" )
      I_Contact( "output"."3号梯上行接触器" )
      I_Contact( "output"."3号梯开门继电器" )
      I_Contact( "output"."3号梯关门继电器" )
      I_Contact( "3号梯开门锁上下行" )
      Coil( "output"."3号梯下行接触器" )
   END_RUNG
   // the same network as SCL:
   "output"."3号梯上行接触器" := "3号梯上行接触器" AND NOT "output"."3号梯下行接触器" AND NOT "output"."3号梯开门继电器" AND NOT "output"."3号梯关门继电器" AND NOT "3号梯开门锁上下行";
   "output"."3号梯下行接触器" := "3号梯下行接触器" AND NOT "output"."3号梯上行接触器" AND NOT "output"."3号梯开门继电器" AND NOT "output"."3号梯关门继电器" AND NOT "3号梯开门锁上下行";
END_REGION

REGION Network 18: 1号梯开关门继电器
   RUNG wire#powerrail
      Contact( "1号梯开门继电器" )
      I_Contact( "output"."1号梯上行接触器" )
      I_Contact( "output"."1号梯下行接触器" )
      I_Contact( "output"."1号梯关门继电器" )
      Coil( "output"."1号梯开门继电器" )
   END_RUNG
   RUNG wire#powerrail
      Contact( "1号梯关门继电器" )
      I_Contact( "output"."1号梯上行接触器" )
      I_Contact( "output"."1号梯下行接触器" )
      I_Contact( "output"."1号梯开门继电器" )
      Coil( "output"."1号梯关门继电器" )
   END_RUNG
   // the same network as SCL:
   "output"."1号梯开门继电器" := "1号梯开门继电器" AND NOT "output"."1号梯上行接触器" AND NOT "output"."1号梯下行接触器" AND NOT "output"."1号梯关门继电器";
   "output"."1号梯关门继电器" := "1号梯关门继电器" AND NOT "output"."1号梯上行接触器" AND NOT "output"."1号梯下行接触器" AND NOT "output"."1号梯开门继电器";
END_REGION

REGION Network 19: 2号梯开关门继电器
   RUNG wire#powerrail
      Contact( "2号梯开门继电器" )
      I_Contact( "output"."2号梯上行接触器" )
      I_Contact( "output"."2号梯下行接触器" )
      I_Contact( "output"."2号梯关门继电器" )
      Coil( "output"."2号梯开门继电器" )
   END_RUNG
   RUNG wire#powerrail
      Contact( "2号梯关门继电器" )
      I_Contact( "output"."2号梯上行接触器" )
      I_Contact( "output"."2号梯下行接触器" )
      I_Contact( "output"."2号梯开门继电器" )
      Coil( "output"."2号梯关门继电器" )
   END_RUNG
   // the same network as SCL:
   "output"."2号梯开门继电器" := "2号梯开门继电器" AND NOT "output"."2号梯上行接触器" AND NOT "output"."2号梯下行接触器" AND NOT "output"."2号梯关门继电器";
   "output"."2号梯关门继电器" := "2号梯关门继电器" AND NOT "output"."2号梯上行接触器" AND NOT "output"."2号梯下行接触器" AND NOT "output"."2号梯开门继电器";
END_REGION

REGION Network 20: 3号梯开关门继电器
   RUNG wire#powerrail
      Contact( "3号梯开门继电器" )
      I_Contact( "output"."3号梯上行接触器" )
      I_Contact( "output"."3号梯下行接触器" )
      I_Contact( "output"."3号梯关门继电器" )
      Coil( "output"."3号梯开门继电器" )
   END_RUNG
   RUNG wire#powerrail
      Contact( "3号梯关门继电器" )
      I_Contact( "output"."3号梯上行接触器" )
      I_Contact( "output"."3号梯下行接触器" )
      I_Contact( "output"."3号梯开门继电器" )
      Coil( "output"."3号梯关门继电器" )
   END_RUNG
   // the same network as SCL:
   "output"."3号梯开门继电器" := "3号梯开门继电器" AND NOT "output"."3号梯上行接触器" AND NOT "output"."3号梯下行接触器" AND NOT "output"."3号梯关门继电器";
   "output"."3号梯关门继电器" := "3号梯关门继电器" AND NOT "output"."3号梯上行接触器" AND NOT "output"."3号梯下行接触器" AND NOT "output"."3号梯开门继电器";
END_REGION

REGION Network 21: 1号梯高低速、减速制动接触器
   RUNG wire#powerrail
      Contact( "1号梯高速运行" )
      I_Contact( "output"."1号梯低速接触器" )
      Coil( "output"."1号梯高速接触器" )
   END_RUNG
   RUNG wire#powerrail
      Contact( "1号梯低速运行" )
      I_Contact( "output"."1号梯高速接触器" )
      Coil( "output"."1号梯低速接触器" )
   END_RUNG
   RUNG wire#powerrail
      Contact( "1号梯1级制动接触器" )
      Coil( "output"."1号梯1级减速制动" )
   END_RUNG
   RUNG wire#powerrail
      Contact( "1号梯2级制动接触器" )
      Coil( "output"."1号梯2级减速制动" )
   END_RUNG
   RUNG wire#powerrail
      Contact( "1号梯3级制动接触器" )
      Coil( "output"."1号梯3级减速制动" )
   END_RUNG
   // the same network as SCL:
   "output"."1号梯高速接触器" := "1号梯高速运行" AND NOT "output"."1号梯低速接触器";
   "output"."1号梯低速接触器" := "1号梯低速运行" AND NOT "output"."1号梯高速接触器";
   "output"."1号梯1级减速制动" := "1号梯1级制动接触器";
   "output"."1号梯2级减速制动" := "1号梯2级制动接触器";
   "output"."1号梯3级减速制动" := "1号梯3级制动接触器";
END_REGION

REGION Network 22: 2号梯高低速、减速制动接触器
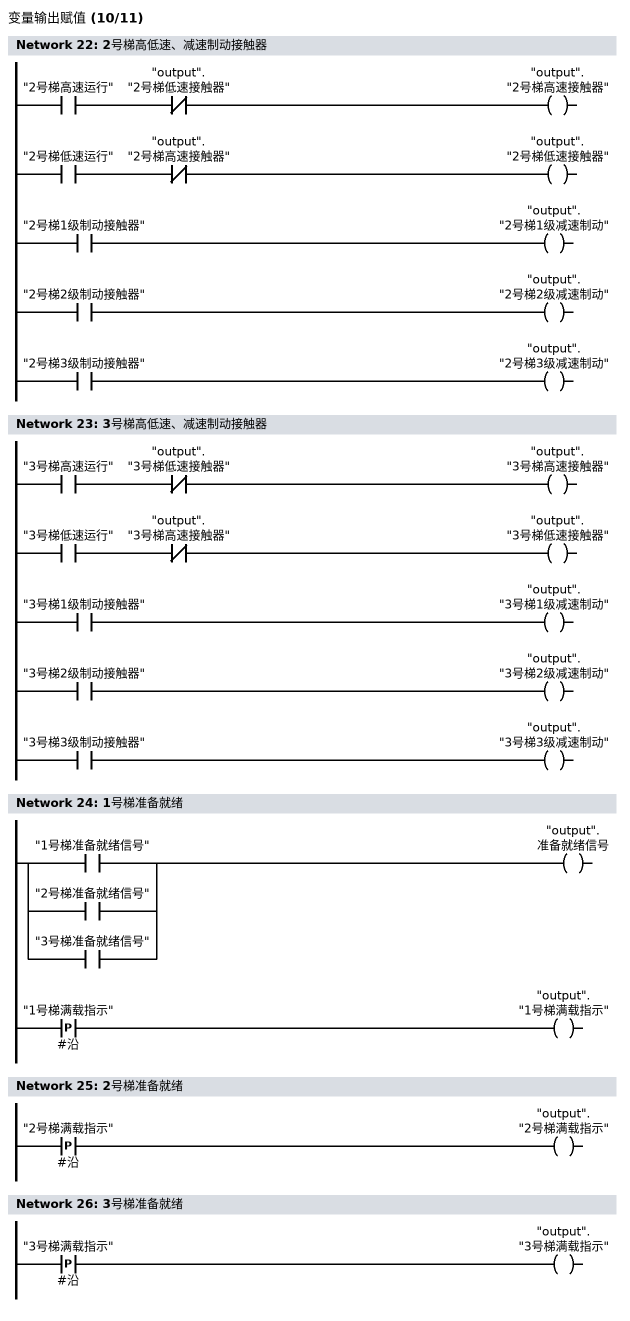
   RUNG wire#powerrail
      Contact( "2号梯高速运行" )
      I_Contact( "output"."2号梯低速接触器" )
      Coil( "output"."2号梯高速接触器" )
   END_RUNG
   RUNG wire#powerrail
      Contact( "2号梯低速运行" )
      I_Contact( "output"."2号梯高速接触器" )
      Coil( "output"."2号梯低速接触器" )
   END_RUNG
   RUNG wire#powerrail
      Contact( "2号梯1级制动接触器" )
      Coil( "output"."2号梯1级减速制动" )
   END_RUNG
   RUNG wire#powerrail
      Contact( "2号梯2级制动接触器" )
      Coil( "output"."2号梯2级减速制动" )
   END_RUNG
   RUNG wire#powerrail
      Contact( "2号梯3级制动接触器" )
      Coil( "output"."2号梯3级减速制动" )
   END_RUNG
   // the same network as SCL:
   "output"."2号梯高速接触器" := "2号梯高速运行" AND NOT "output"."2号梯低速接触器";
   "output"."2号梯低速接触器" := "2号梯低速运行" AND NOT "output"."2号梯高速接触器";
   "output"."2号梯1级减速制动" := "2号梯1级制动接触器";
   "output"."2号梯2级减速制动" := "2号梯2级制动接触器";
   "output"."2号梯3级减速制动" := "2号梯3级制动接触器";
END_REGION

REGION Network 23: 3号梯高低速、减速制动接触器
   RUNG wire#powerrail
      Contact( "3号梯高速运行" )
      I_Contact( "output"."3号梯低速接触器" )
      Coil( "output"."3号梯高速接触器" )
   END_RUNG
   RUNG wire#powerrail
      Contact( "3号梯低速运行" )
      I_Contact( "output"."3号梯高速接触器" )
      Coil( "output"."3号梯低速接触器" )
   END_RUNG
   RUNG wire#powerrail
      Contact( "3号梯1级制动接触器" )
      Coil( "output"."3号梯1级减速制动" )
   END_RUNG
   RUNG wire#powerrail
      Contact( "3号梯2级制动接触器" )
      Coil( "output"."3号梯2级减速制动" )
   END_RUNG
   RUNG wire#powerrail
      Contact( "3号梯3级制动接触器" )
      Coil( "output"."3号梯3级减速制动" )
   END_RUNG
   // the same network as SCL:
   "output"."3号梯高速接触器" := "3号梯高速运行" AND NOT "output"."3号梯低速接触器";
   "output"."3号梯低速接触器" := "3号梯低速运行" AND NOT "output"."3号梯高速接触器";
   "output"."3号梯1级减速制动" := "3号梯1级制动接触器";
   "output"."3号梯2级减速制动" := "3号梯2级制动接触器";
   "output"."3号梯3级减速制动" := "3号梯3级制动接触器";
END_REGION

REGION Network 24: 1号梯准备就绪
   RUNG wire#powerrail
      Contact( "1号梯准备就绪信号" )
      wire#w1
      Coil( "output".准备就绪信号 )
   END_RUNG
   RUNG wire#powerrail
      Contact( "2号梯准备就绪信号" )
   END_RUNG wire#w1
   RUNG wire#powerrail
      Contact( "3号梯准备就绪信号" )
   END_RUNG wire#w1
   RUNG wire#powerrail
      P_Contact(operand := "1号梯满载指示", bit := #沿)
      Coil( "output"."1号梯满载指示" )
   END_RUNG
   // the same network as SCL:
   "output".准备就绪信号 := "1号梯准备就绪信号" OR "2号梯准备就绪信号" OR "3号梯准备就绪信号";
   #_w1 := "1号梯满载指示" AND NOT #沿;   // rising edge of "1号梯满载指示"
   #沿 := "1号梯满载指示";
   "output"."1号梯满载指示" := #_w1;
END_REGION

REGION Network 25: 2号梯准备就绪
   RUNG wire#powerrail
      P_Contact(operand := "2号梯满载指示", bit := #沿)
      Coil( "output"."2号梯满载指示" )
   END_RUNG
   // the same network as SCL:
   #_w1 := "2号梯满载指示" AND NOT #沿;   // rising edge of "2号梯满载指示"
   #沿 := "2号梯满载指示";
   "output"."2号梯满载指示" := #_w1;
END_REGION

REGION Network 26: 3号梯准备就绪
   RUNG wire#powerrail
      P_Contact(operand := "3号梯满载指示", bit := #沿)
      Coil( "output"."3号梯满载指示" )
   END_RUNG
   // the same network as SCL:
   #_w1 := "3号梯满载指示" AND NOT #沿;   // rising edge of "3号梯满载指示"
   #沿 := "3号梯满载指示";
   "output"."3号梯满载指示" := #_w1;
END_REGION

REGION Network 27: 电机启动
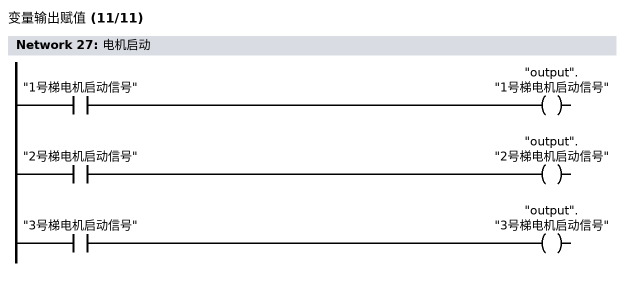
   RUNG wire#powerrail
      Contact( "1号梯电机启动信号" )
      Coil( "output"."1号梯电机启动信号" )
   END_RUNG
   RUNG wire#powerrail
      Contact( "2号梯电机启动信号" )
      Coil( "output"."2号梯电机启动信号" )
   END_RUNG
   RUNG wire#powerrail
      Contact( "3号梯电机启动信号" )
      Coil( "output"."3号梯电机启动信号" )
   END_RUNG
   // the same network as SCL:
   "output"."1号梯电机启动信号" := "1号梯电机启动信号";
   "output"."2号梯电机启动信号" := "2号梯电机启动信号";
   "output"."3号梯电机启动信号" := "3号梯电机启动信号";
END_REGION
END_FUNCTION

FUNCTION "变量输入赋值" : Void   // FC3, LAD
{ S7_Optimized_Access := 'TRUE' }
VERSION : 0.1
   VAR_TEMP   // added for the SCL form of the ladder/FBD networks
      _w1 : Bool;
      _w2 : Bool;
      _w3 : Bool;
      _w4 : Bool;
   END_VAR
BEGIN

REGION Network 1: 1号梯内呼按钮
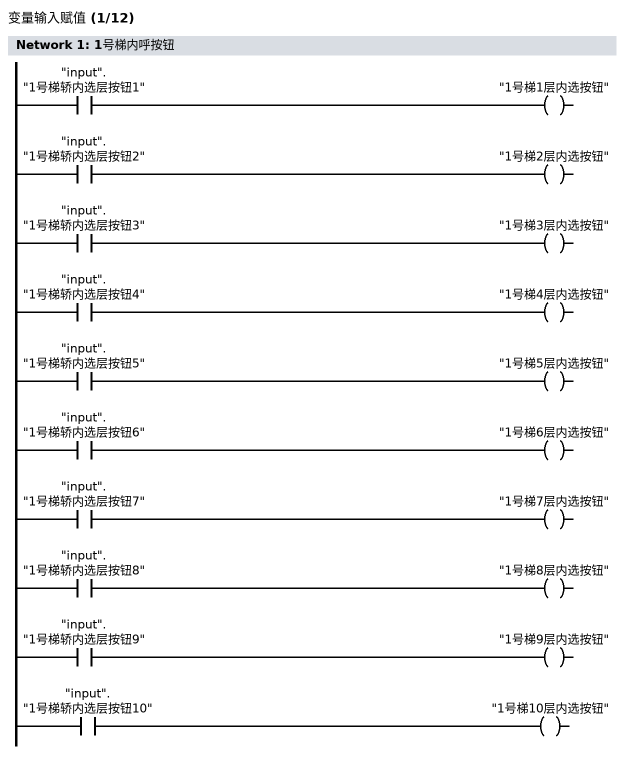
   RUNG wire#powerrail
      Contact( "input"."1号梯轿内选层按钮1" )
      Coil( "1号梯1层内选按钮" )
   END_RUNG
   RUNG wire#powerrail
      Contact( "input"."1号梯轿内选层按钮2" )
      Coil( "1号梯2层内选按钮" )
   END_RUNG
   RUNG wire#powerrail
      Contact( "input"."1号梯轿内选层按钮3" )
      Coil( "1号梯3层内选按钮" )
   END_RUNG
   RUNG wire#powerrail
      Contact( "input"."1号梯轿内选层按钮4" )
      Coil( "1号梯4层内选按钮" )
   END_RUNG
   RUNG wire#powerrail
      Contact( "input"."1号梯轿内选层按钮5" )
      Coil( "1号梯5层内选按钮" )
   END_RUNG
   RUNG wire#powerrail
      Contact( "input"."1号梯轿内选层按钮6" )
      Coil( "1号梯6层内选按钮" )
   END_RUNG
   RUNG wire#powerrail
      Contact( "input"."1号梯轿内选层按钮7" )
      Coil( "1号梯7层内选按钮" )
   END_RUNG
   RUNG wire#powerrail
      Contact( "input"."1号梯轿内选层按钮8" )
      Coil( "1号梯8层内选按钮" )
   END_RUNG
   RUNG wire#powerrail
      Contact( "input"."1号梯轿内选层按钮9" )
      Coil( "1号梯9层内选按钮" )
   END_RUNG
   RUNG wire#powerrail
      Contact( "input"."1号梯轿内选层按钮10" )
      Coil( "1号梯10层内选按钮" )
   END_RUNG
   // the same network as SCL:
   "1号梯1层内选按钮" := "input"."1号梯轿内选层按钮1";
   "1号梯2层内选按钮" := "input"."1号梯轿内选层按钮2";
   "1号梯3层内选按钮" := "input"."1号梯轿内选层按钮3";
   "1号梯4层内选按钮" := "input"."1号梯轿内选层按钮4";
   "1号梯5层内选按钮" := "input"."1号梯轿内选层按钮5";
   "1号梯6层内选按钮" := "input"."1号梯轿内选层按钮6";
   "1号梯7层内选按钮" := "input"."1号梯轿内选层按钮7";
   "1号梯8层内选按钮" := "input"."1号梯轿内选层按钮8";
   "1号梯9层内选按钮" := "input"."1号梯轿内选层按钮9";
   "1号梯10层内选按钮" := "input"."1号梯轿内选层按钮10";
END_REGION

REGION Network 2: 2号梯内呼按钮
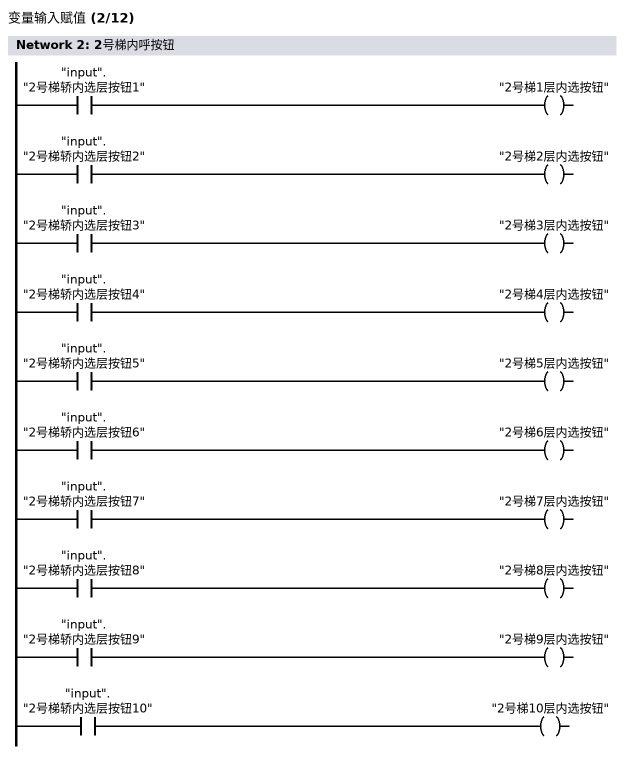
   RUNG wire#powerrail
      Contact( "input"."2号梯轿内选层按钮1" )
      Coil( "2号梯1层内选按钮" )
   END_RUNG
   RUNG wire#powerrail
      Contact( "input"."2号梯轿内选层按钮2" )
      Coil( "2号梯2层内选按钮" )
   END_RUNG
   RUNG wire#powerrail
      Contact( "input"."2号梯轿内选层按钮3" )
      Coil( "2号梯3层内选按钮" )
   END_RUNG
   RUNG wire#powerrail
      Contact( "input"."2号梯轿内选层按钮4" )
      Coil( "2号梯4层内选按钮" )
   END_RUNG
   RUNG wire#powerrail
      Contact( "input"."2号梯轿内选层按钮5" )
      Coil( "2号梯5层内选按钮" )
   END_RUNG
   RUNG wire#powerrail
      Contact( "input"."2号梯轿内选层按钮6" )
      Coil( "2号梯6层内选按钮" )
   END_RUNG
   RUNG wire#powerrail
      Contact( "input"."2号梯轿内选层按钮7" )
      Coil( "2号梯7层内选按钮" )
   END_RUNG
   RUNG wire#powerrail
      Contact( "input"."2号梯轿内选层按钮8" )
      Coil( "2号梯8层内选按钮" )
   END_RUNG
   RUNG wire#powerrail
      Contact( "input"."2号梯轿内选层按钮9" )
      Coil( "2号梯9层内选按钮" )
   END_RUNG
   RUNG wire#powerrail
      Contact( "input"."2号梯轿内选层按钮10" )
      Coil( "2号梯10层内选按钮" )
   END_RUNG
   // the same network as SCL:
   "2号梯1层内选按钮" := "input"."2号梯轿内选层按钮1";
   "2号梯2层内选按钮" := "input"."2号梯轿内选层按钮2";
   "2号梯3层内选按钮" := "input"."2号梯轿内选层按钮3";
   "2号梯4层内选按钮" := "input"."2号梯轿内选层按钮4";
   "2号梯5层内选按钮" := "input"."2号梯轿内选层按钮5";
   "2号梯6层内选按钮" := "input"."2号梯轿内选层按钮6";
   "2号梯7层内选按钮" := "input"."2号梯轿内选层按钮7";
   "2号梯8层内选按钮" := "input"."2号梯轿内选层按钮8";
   "2号梯9层内选按钮" := "input"."2号梯轿内选层按钮9";
   "2号梯10层内选按钮" := "input"."2号梯轿内选层按钮10";
END_REGION

REGION Network 3: 3号梯内呼按钮
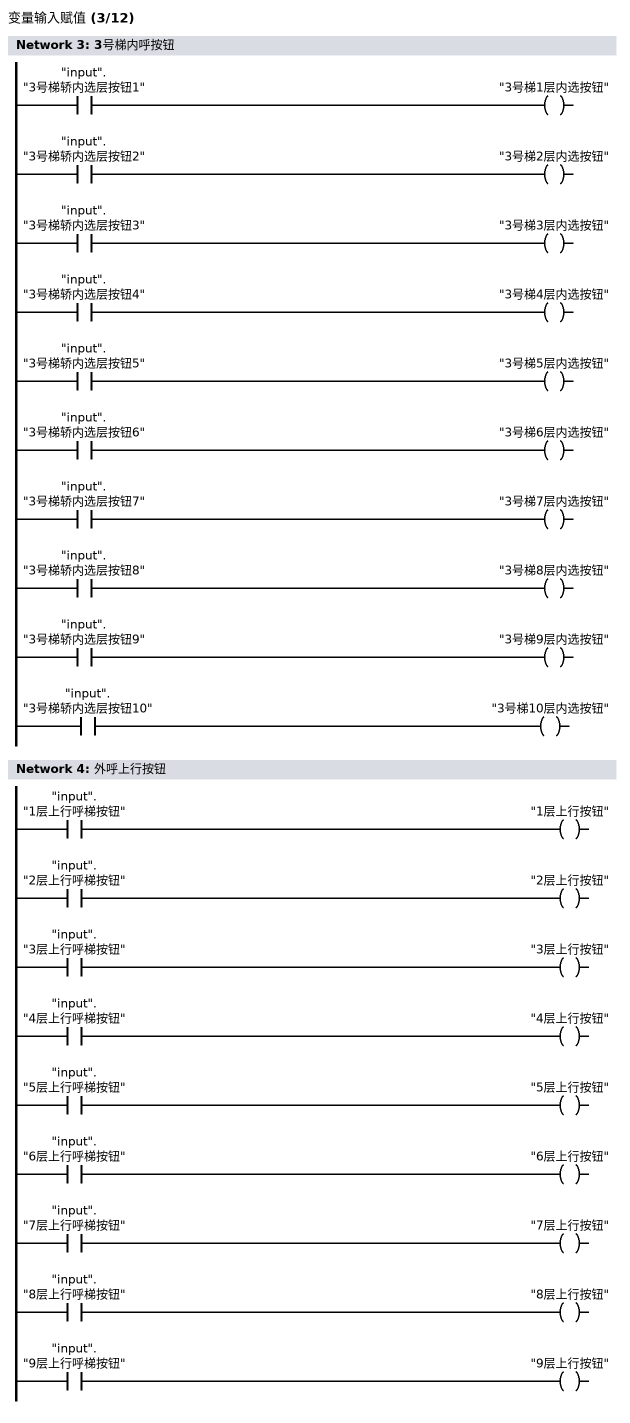
   RUNG wire#powerrail
      Contact( "input"."3号梯轿内选层按钮1" )
      Coil( "3号梯1层内选按钮" )
   END_RUNG
   RUNG wire#powerrail
      Contact( "input"."3号梯轿内选层按钮2" )
      Coil( "3号梯2层内选按钮" )
   END_RUNG
   RUNG wire#powerrail
      Contact( "input"."3号梯轿内选层按钮3" )
      Coil( "3号梯3层内选按钮" )
   END_RUNG
   RUNG wire#powerrail
      Contact( "input"."3号梯轿内选层按钮4" )
      Coil( "3号梯4层内选按钮" )
   END_RUNG
   RUNG wire#powerrail
      Contact( "input"."3号梯轿内选层按钮5" )
      Coil( "3号梯5层内选按钮" )
   END_RUNG
   RUNG wire#powerrail
      Contact( "input"."3号梯轿内选层按钮6" )
      Coil( "3号梯6层内选按钮" )
   END_RUNG
   RUNG wire#powerrail
      Contact( "input"."3号梯轿内选层按钮7" )
      Coil( "3号梯7层内选按钮" )
   END_RUNG
   RUNG wire#powerrail
      Contact( "input"."3号梯轿内选层按钮8" )
      Coil( "3号梯8层内选按钮" )
   END_RUNG
   RUNG wire#powerrail
      Contact( "input"."3号梯轿内选层按钮9" )
      Coil( "3号梯9层内选按钮" )
   END_RUNG
   RUNG wire#powerrail
      Contact( "input"."3号梯轿内选层按钮10" )
      Coil( "3号梯10层内选按钮" )
   END_RUNG
   // the same network as SCL:
   "3号梯1层内选按钮" := "input"."3号梯轿内选层按钮1";
   "3号梯2层内选按钮" := "input"."3号梯轿内选层按钮2";
   "3号梯3层内选按钮" := "input"."3号梯轿内选层按钮3";
   "3号梯4层内选按钮" := "input"."3号梯轿内选层按钮4";
   "3号梯5层内选按钮" := "input"."3号梯轿内选层按钮5";
   "3号梯6层内选按钮" := "input"."3号梯轿内选层按钮6";
   "3号梯7层内选按钮" := "input"."3号梯轿内选层按钮7";
   "3号梯8层内选按钮" := "input"."3号梯轿内选层按钮8";
   "3号梯9层内选按钮" := "input"."3号梯轿内选层按钮9";
   "3号梯10层内选按钮" := "input"."3号梯轿内选层按钮10";
END_REGION

REGION Network 4: 外呼上行按钮
   RUNG wire#powerrail
      Contact( "input"."1层上行呼梯按钮" )
      Coil( "1层上行按钮" )
   END_RUNG
   RUNG wire#powerrail
      Contact( "input"."2层上行呼梯按钮" )
      Coil( "2层上行按钮" )
   END_RUNG
   RUNG wire#powerrail
      Contact( "input"."3层上行呼梯按钮" )
      Coil( "3层上行按钮" )
   END_RUNG
   RUNG wire#powerrail
      Contact( "input"."4层上行呼梯按钮" )
      Coil( "4层上行按钮" )
   END_RUNG
   RUNG wire#powerrail
      Contact( "input"."5层上行呼梯按钮" )
      Coil( "5层上行按钮" )
   END_RUNG
   RUNG wire#powerrail
      Contact( "input"."6层上行呼梯按钮" )
      Coil( "6层上行按钮" )
   END_RUNG
   RUNG wire#powerrail
      Contact( "input"."7层上行呼梯按钮" )
      Coil( "7层上行按钮" )
   END_RUNG
   RUNG wire#powerrail
      Contact( "input"."8层上行呼梯按钮" )
      Coil( "8层上行按钮" )
   END_RUNG
   RUNG wire#powerrail
      Contact( "input"."9层上行呼梯按钮" )
      Coil( "9层上行按钮" )
   END_RUNG
   // the same network as SCL:
   "1层上行按钮" := "input"."1层上行呼梯按钮";
   "2层上行按钮" := "input"."2层上行呼梯按钮";
   "3层上行按钮" := "input"."3层上行呼梯按钮";
   "4层上行按钮" := "input"."4层上行呼梯按钮";
   "5层上行按钮" := "input"."5层上行呼梯按钮";
   "6层上行按钮" := "input"."6层上行呼梯按钮";
   "7层上行按钮" := "input"."7层上行呼梯按钮";
   "8层上行按钮" := "input"."8层上行呼梯按钮";
   "9层上行按钮" := "input"."9层上行呼梯按钮";
END_REGION

REGION Network 5: 外呼下行按钮
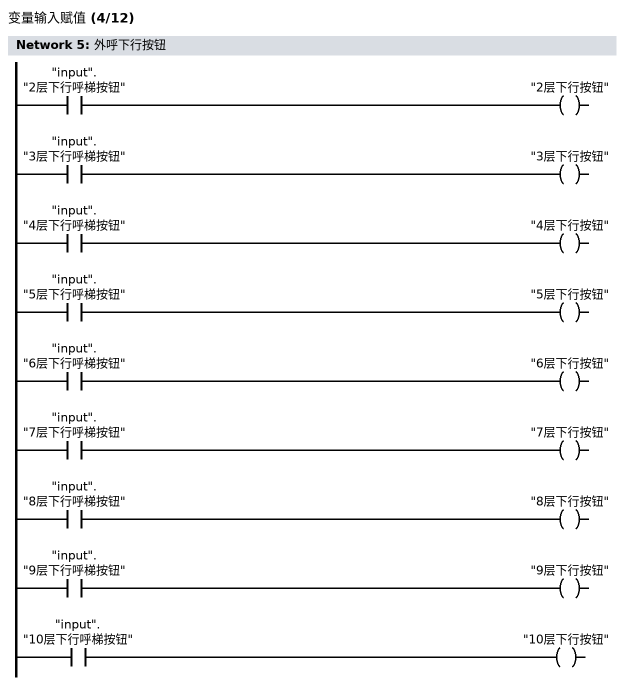
   RUNG wire#powerrail
      Contact( "input"."2层下行呼梯按钮" )
      Coil( "2层下行按钮" )
   END_RUNG
   RUNG wire#powerrail
      Contact( "input"."3层下行呼梯按钮" )
      Coil( "3层下行按钮" )
   END_RUNG
   RUNG wire#powerrail
      Contact( "input"."4层下行呼梯按钮" )
      Coil( "4层下行按钮" )
   END_RUNG
   RUNG wire#powerrail
      Contact( "input"."5层下行呼梯按钮" )
      Coil( "5层下行按钮" )
   END_RUNG
   RUNG wire#powerrail
      Contact( "input"."6层下行呼梯按钮" )
      Coil( "6层下行按钮" )
   END_RUNG
   RUNG wire#powerrail
      Contact( "input"."7层下行呼梯按钮" )
      Coil( "7层下行按钮" )
   END_RUNG
   RUNG wire#powerrail
      Contact( "input"."8层下行呼梯按钮" )
      Coil( "8层下行按钮" )
   END_RUNG
   RUNG wire#powerrail
      Contact( "input"."9层下行呼梯按钮" )
      Coil( "9层下行按钮" )
   END_RUNG
   RUNG wire#powerrail
      Contact( "input"."10层下行呼梯按钮" )
      Coil( "10层下行按钮" )
   END_RUNG
   // the same network as SCL:
   "2层下行按钮" := "input"."2层下行呼梯按钮";
   "3层下行按钮" := "input"."3层下行呼梯按钮";
   "4层下行按钮" := "input"."4层下行呼梯按钮";
   "5层下行按钮" := "input"."5层下行呼梯按钮";
   "6层下行按钮" := "input"."6层下行呼梯按钮";
   "7层下行按钮" := "input"."7层下行呼梯按钮";
   "8层下行按钮" := "input"."8层下行呼梯按钮";
   "9层下行按钮" := "input"."9层下行呼梯按钮";
   "10层下行按钮" := "input"."10层下行呼梯按钮";
END_REGION

REGION Network 6: 1号梯开关门、光幕、载重、检修信号
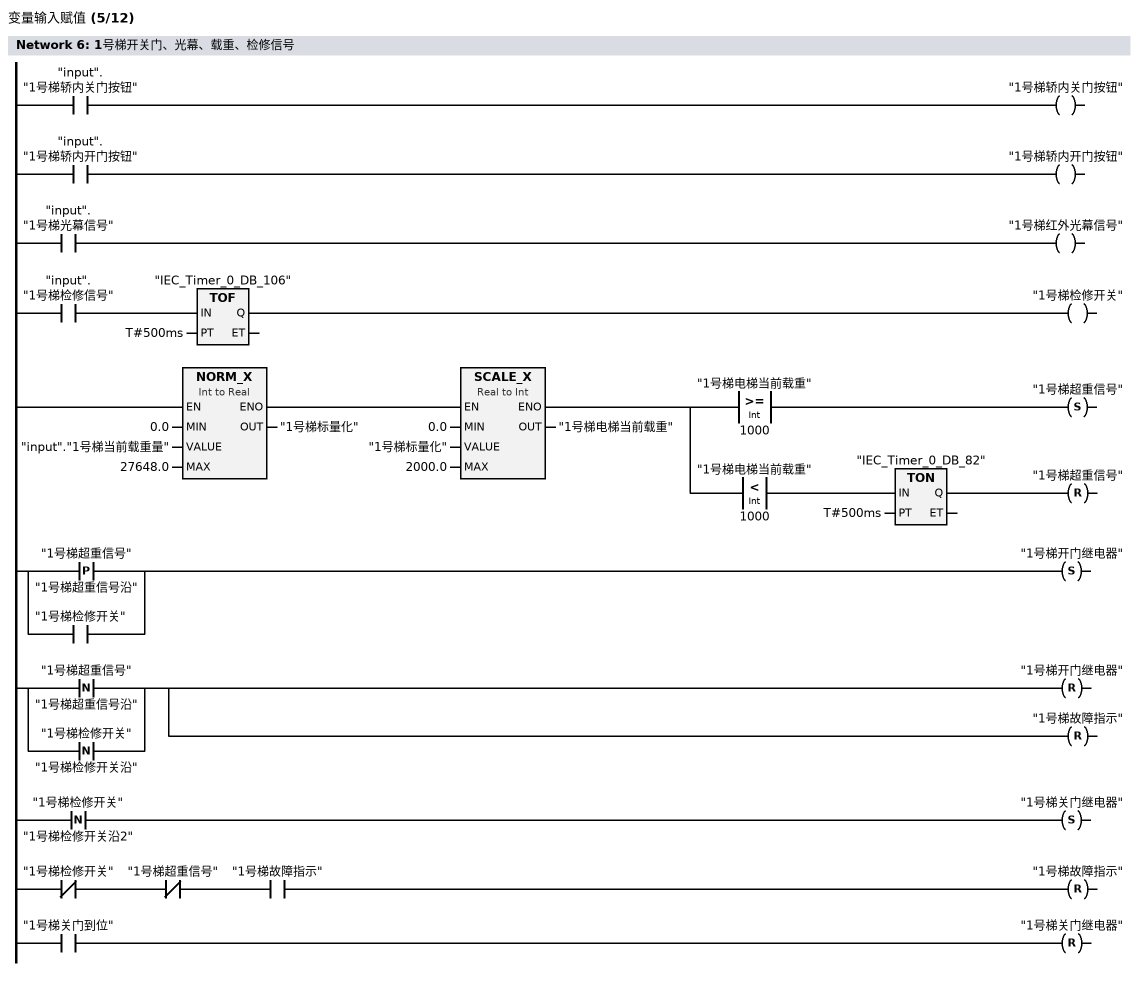
   "1号梯轿内关门按钮" := "input"."1号梯轿内关门按钮";
   "1号梯轿内开门按钮" := "input"."1号梯轿内开门按钮";
   "1号梯红外光幕信号" := "input"."1号梯光幕信号";
   "IEC_Timer_0_DB_106".TOF(IN := "input"."1号梯检修信号", PT := T#500ms);
   "1号梯检修开关" := "IEC_Timer_0_DB_106".Q;
   "1号梯标量化" := NORM_X(MIN := 0.0, VALUE := "input"."1号梯当前载重量", MAX := 27648.0);
   "1号梯电梯当前载重" := SCALE_X(MIN := 0.0, VALUE := "1号梯标量化", MAX := 2000.0);
   IF "1号梯电梯当前载重" >= 1000 THEN "1号梯超重信号" := TRUE; END_IF;
   "IEC_Timer_0_DB_82".TON(IN := "1号梯电梯当前载重" < 1000, PT := T#500ms);
   IF "IEC_Timer_0_DB_82".Q THEN "1号梯超重信号" := FALSE; END_IF;
   #_w1 := "1号梯超重信号" AND NOT "1号梯超重信号沿";   // rising edge of "1号梯超重信号"
   "1号梯超重信号沿" := "1号梯超重信号";
   IF #_w1 OR "1号梯检修开关" THEN "1号梯开门继电器" := TRUE; END_IF;
   #_w2 := NOT "1号梯超重信号" AND "1号梯超重信号沿";   // falling edge of "1号梯超重信号"
   "1号梯超重信号沿" := "1号梯超重信号";
   #_w3 := NOT "1号梯检修开关" AND "1号梯检修开关沿";   // falling edge of "1号梯检修开关"
   "1号梯检修开关沿" := "1号梯检修开关";
   IF #_w2 OR #_w3 THEN
       "1号梯开门继电器" := FALSE;
       "1号梯故障指示" := FALSE;
   END_IF;
   #_w4 := NOT "1号梯检修开关" AND "1号梯检修开关沿2";   // falling edge of "1号梯检修开关"
   "1号梯检修开关沿2" := "1号梯检修开关";
   IF #_w4 THEN "1号梯关门继电器" := TRUE; END_IF;
   IF NOT "1号梯检修开关" AND NOT "1号梯超重信号" AND "1号梯故障指示" THEN "1号梯故障指示" := FALSE; END_IF;
   IF "1号梯关门到位" THEN "1号梯关门继电器" := FALSE; END_IF;
END_REGION

REGION Network 7: 2号梯开关门、光幕、载重、检修信号
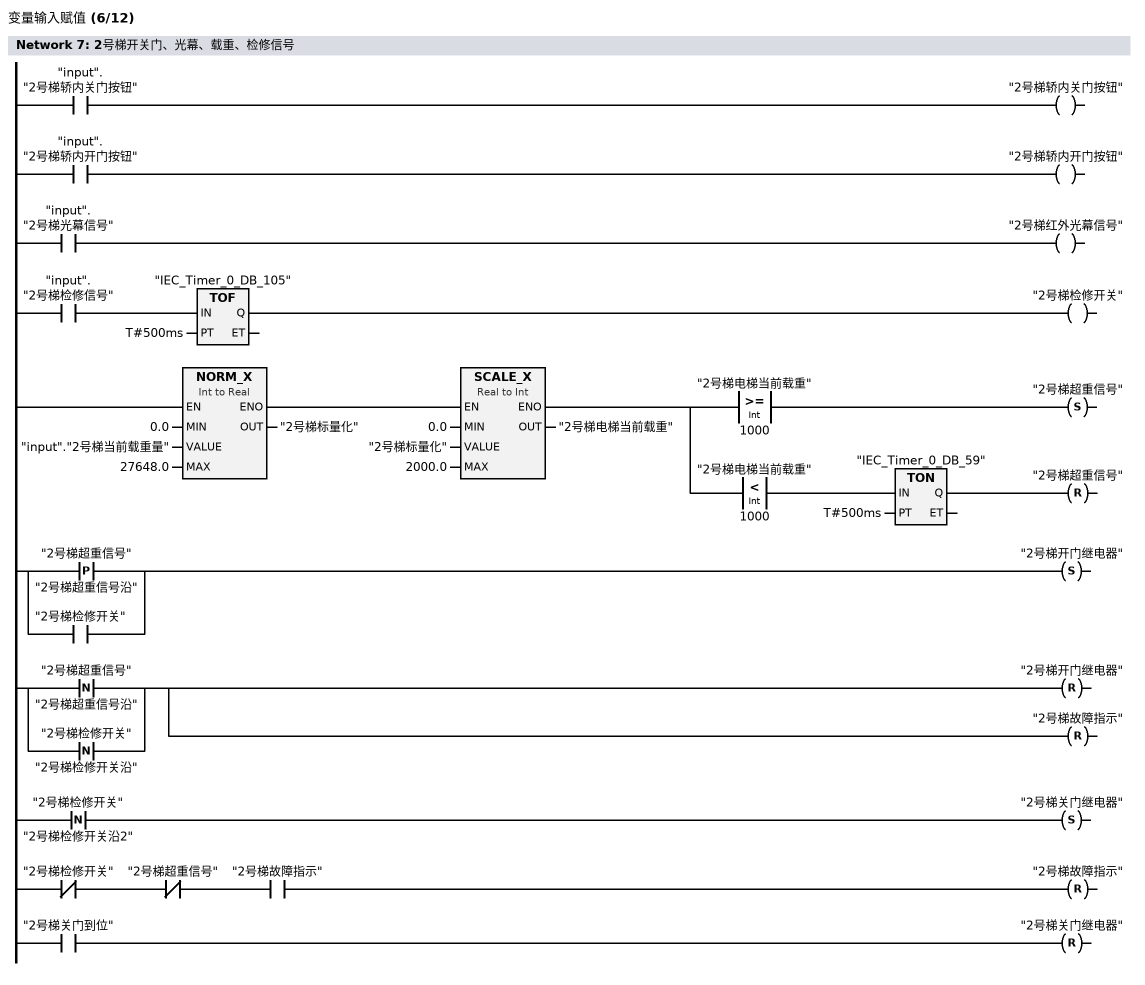
   "2号梯轿内关门按钮" := "input"."2号梯轿内关门按钮";
   "2号梯轿内开门按钮" := "input"."2号梯轿内开门按钮";
   "2号梯红外光幕信号" := "input"."2号梯光幕信号";
   "IEC_Timer_0_DB_105".TOF(IN := "input"."2号梯检修信号", PT := T#500ms);
   "2号梯检修开关" := "IEC_Timer_0_DB_105".Q;
   "2号梯标量化" := NORM_X(MIN := 0.0, VALUE := "input"."2号梯当前载重量", MAX := 27648.0);
   "2号梯电梯当前载重" := SCALE_X(MIN := 0.0, VALUE := "2号梯标量化", MAX := 2000.0);
   IF "2号梯电梯当前载重" >= 1000 THEN "2号梯超重信号" := TRUE; END_IF;
   "IEC_Timer_0_DB_59".TON(IN := "2号梯电梯当前载重" < 1000, PT := T#500ms);
   IF "IEC_Timer_0_DB_59".Q THEN "2号梯超重信号" := FALSE; END_IF;
   #_w1 := "2号梯超重信号" AND NOT "2号梯超重信号沿";   // rising edge of "2号梯超重信号"
   "2号梯超重信号沿" := "2号梯超重信号";
   IF #_w1 OR "2号梯检修开关" THEN "2号梯开门继电器" := TRUE; END_IF;
   #_w2 := NOT "2号梯超重信号" AND "2号梯超重信号沿";   // falling edge of "2号梯超重信号"
   "2号梯超重信号沿" := "2号梯超重信号";
   #_w3 := NOT "2号梯检修开关" AND "2号梯检修开关沿";   // falling edge of "2号梯检修开关"
   "2号梯检修开关沿" := "2号梯检修开关";
   IF #_w2 OR #_w3 THEN
       "2号梯开门继电器" := FALSE;
       "2号梯故障指示" := FALSE;
   END_IF;
   #_w4 := NOT "2号梯检修开关" AND "2号梯检修开关沿2";   // falling edge of "2号梯检修开关"
   "2号梯检修开关沿2" := "2号梯检修开关";
   IF #_w4 THEN "2号梯关门继电器" := TRUE; END_IF;
   IF NOT "2号梯检修开关" AND NOT "2号梯超重信号" AND "2号梯故障指示" THEN "2号梯故障指示" := FALSE; END_IF;
   IF "2号梯关门到位" THEN "2号梯关门继电器" := FALSE; END_IF;
END_REGION

REGION Network 8: 3号梯开关门、光幕、载重、检修信号
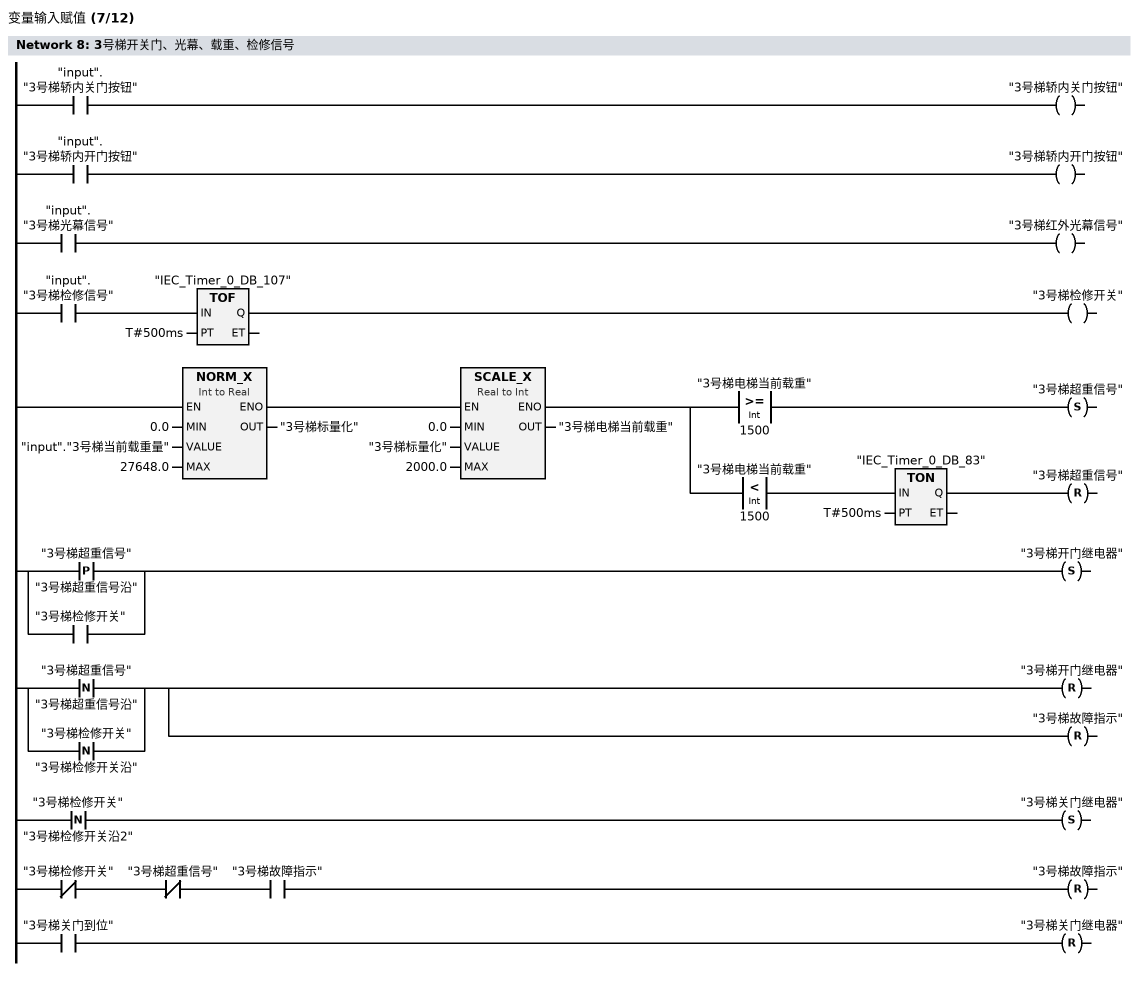
   "3号梯轿内关门按钮" := "input"."3号梯轿内关门按钮";
   "3号梯轿内开门按钮" := "input"."3号梯轿内开门按钮";
   "3号梯红外光幕信号" := "input"."3号梯光幕信号";
   "IEC_Timer_0_DB_107".TOF(IN := "input"."3号梯检修信号", PT := T#500ms);
   "3号梯检修开关" := "IEC_Timer_0_DB_107".Q;
   "3号梯标量化" := NORM_X(MIN := 0.0, VALUE := "input"."3号梯当前载重量", MAX := 27648.0);
   "3号梯电梯当前载重" := SCALE_X(MIN := 0.0, VALUE := "3号梯标量化", MAX := 2000.0);
   IF "3号梯电梯当前载重" >= 1500 THEN "3号梯超重信号" := TRUE; END_IF;
   "IEC_Timer_0_DB_83".TON(IN := "3号梯电梯当前载重" < 1500, PT := T#500ms);
   IF "IEC_Timer_0_DB_83".Q THEN "3号梯超重信号" := FALSE; END_IF;
   #_w1 := "3号梯超重信号" AND NOT "3号梯超重信号沿";   // rising edge of "3号梯超重信号"
   "3号梯超重信号沿" := "3号梯超重信号";
   IF #_w1 OR "3号梯检修开关" THEN "3号梯开门继电器" := TRUE; END_IF;
   #_w2 := NOT "3号梯超重信号" AND "3号梯超重信号沿";   // falling edge of "3号梯超重信号"
   "3号梯超重信号沿" := "3号梯超重信号";
   #_w3 := NOT "3号梯检修开关" AND "3号梯检修开关沿";   // falling edge of "3号梯检修开关"
   "3号梯检修开关沿" := "3号梯检修开关";
   IF #_w2 OR #_w3 THEN
       "3号梯开门继电器" := FALSE;
       "3号梯故障指示" := FALSE;
   END_IF;
   #_w4 := NOT "3号梯检修开关" AND "3号梯检修开关沿2";   // falling edge of "3号梯检修开关"
   "3号梯检修开关沿2" := "3号梯检修开关";
   IF #_w4 THEN "3号梯关门继电器" := TRUE; END_IF;
   IF NOT "3号梯检修开关" AND NOT "3号梯超重信号" AND "3号梯故障指示" THEN "3号梯故障指示" := FALSE; END_IF;
   IF "3号梯关门到位" THEN "3号梯关门继电器" := FALSE; END_IF;
END_REGION

REGION Network 9: 1号梯门锁信号
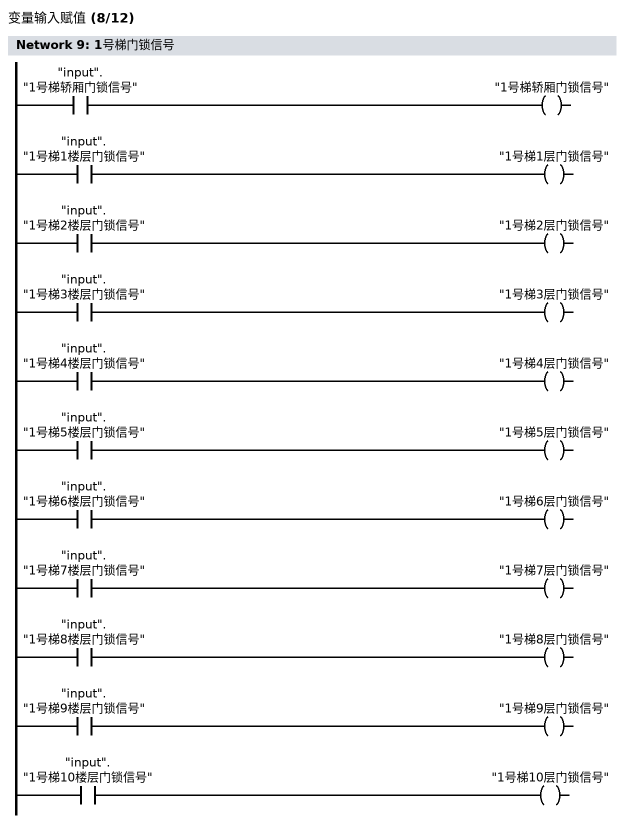
   RUNG wire#powerrail
      Contact( "input"."1号梯轿厢门锁信号" )
      Coil( "1号梯轿厢门锁信号" )
   END_RUNG
   RUNG wire#powerrail
      Contact( "input"."1号梯1楼层门锁信号" )
      Coil( "1号梯1层门锁信号" )
   END_RUNG
   RUNG wire#powerrail
      Contact( "input"."1号梯2楼层门锁信号" )
      Coil( "1号梯2层门锁信号" )
   END_RUNG
   RUNG wire#powerrail
      Contact( "input"."1号梯3楼层门锁信号" )
      Coil( "1号梯3层门锁信号" )
   END_RUNG
   RUNG wire#powerrail
      Contact( "input"."1号梯4楼层门锁信号" )
      Coil( "1号梯4层门锁信号" )
   END_RUNG
   RUNG wire#powerrail
      Contact( "input"."1号梯5楼层门锁信号" )
      Coil( "1号梯5层门锁信号" )
   END_RUNG
   RUNG wire#powerrail
      Contact( "input"."1号梯6楼层门锁信号" )
      Coil( "1号梯6层门锁信号" )
   END_RUNG
   RUNG wire#powerrail
      Contact( "input"."1号梯7楼层门锁信号" )
      Coil( "1号梯7层门锁信号" )
   END_RUNG
   RUNG wire#powerrail
      Contact( "input"."1号梯8楼层门锁信号" )
      Coil( "1号梯8层门锁信号" )
   END_RUNG
   RUNG wire#powerrail
      Contact( "input"."1号梯9楼层门锁信号" )
      Coil( "1号梯9层门锁信号" )
   END_RUNG
   RUNG wire#powerrail
      Contact( "input"."1号梯10楼层门锁信号" )
      Coil( "1号梯10层门锁信号" )
   END_RUNG
   // the same network as SCL:
   "1号梯轿厢门锁信号" := "input"."1号梯轿厢门锁信号";
   "1号梯1层门锁信号" := "input"."1号梯1楼层门锁信号";
   "1号梯2层门锁信号" := "input"."1号梯2楼层门锁信号";
   "1号梯3层门锁信号" := "input"."1号梯3楼层门锁信号";
   "1号梯4层门锁信号" := "input"."1号梯4楼层门锁信号";
   "1号梯5层门锁信号" := "input"."1号梯5楼层门锁信号";
   "1号梯6层门锁信号" := "input"."1号梯6楼层门锁信号";
   "1号梯7层门锁信号" := "input"."1号梯7楼层门锁信号";
   "1号梯8层门锁信号" := "input"."1号梯8楼层门锁信号";
   "1号梯9层门锁信号" := "input"."1号梯9楼层门锁信号";
   "1号梯10层门锁信号" := "input"."1号梯10楼层门锁信号";
END_REGION

REGION Network 10: 2号梯门锁信号
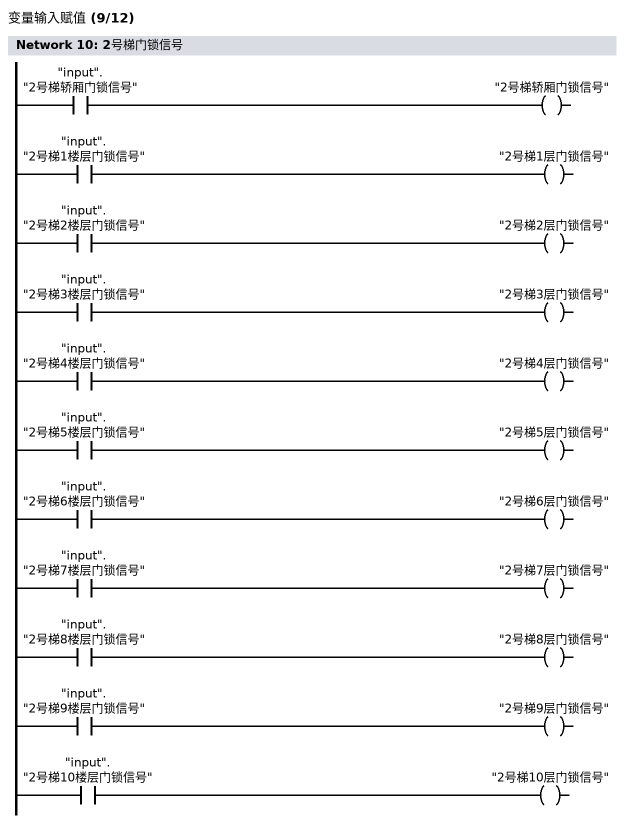
   RUNG wire#powerrail
      Contact( "input"."2号梯轿厢门锁信号" )
      Coil( "2号梯轿厢门锁信号" )
   END_RUNG
   RUNG wire#powerrail
      Contact( "input"."2号梯1楼层门锁信号" )
      Coil( "2号梯1层门锁信号" )
   END_RUNG
   RUNG wire#powerrail
      Contact( "input"."2号梯2楼层门锁信号" )
      Coil( "2号梯2层门锁信号" )
   END_RUNG
   RUNG wire#powerrail
      Contact( "input"."2号梯3楼层门锁信号" )
      Coil( "2号梯3层门锁信号" )
   END_RUNG
   RUNG wire#powerrail
      Contact( "input"."2号梯4楼层门锁信号" )
      Coil( "2号梯4层门锁信号" )
   END_RUNG
   RUNG wire#powerrail
      Contact( "input"."2号梯5楼层门锁信号" )
      Coil( "2号梯5层门锁信号" )
   END_RUNG
   RUNG wire#powerrail
      Contact( "input"."2号梯6楼层门锁信号" )
      Coil( "2号梯6层门锁信号" )
   END_RUNG
   RUNG wire#powerrail
      Contact( "input"."2号梯7楼层门锁信号" )
      Coil( "2号梯7层门锁信号" )
   END_RUNG
   RUNG wire#powerrail
      Contact( "input"."2号梯8楼层门锁信号" )
      Coil( "2号梯8层门锁信号" )
   END_RUNG
   RUNG wire#powerrail
      Contact( "input"."2号梯9楼层门锁信号" )
      Coil( "2号梯9层门锁信号" )
   END_RUNG
   RUNG wire#powerrail
      Contact( "input"."2号梯10楼层门锁信号" )
      Coil( "2号梯10层门锁信号" )
   END_RUNG
   // the same network as SCL:
   "2号梯轿厢门锁信号" := "input"."2号梯轿厢门锁信号";
   "2号梯1层门锁信号" := "input"."2号梯1楼层门锁信号";
   "2号梯2层门锁信号" := "input"."2号梯2楼层门锁信号";
   "2号梯3层门锁信号" := "input"."2号梯3楼层门锁信号";
   "2号梯4层门锁信号" := "input"."2号梯4楼层门锁信号";
   "2号梯5层门锁信号" := "input"."2号梯5楼层门锁信号";
   "2号梯6层门锁信号" := "input"."2号梯6楼层门锁信号";
   "2号梯7层门锁信号" := "input"."2号梯7楼层门锁信号";
   "2号梯8层门锁信号" := "input"."2号梯8楼层门锁信号";
   "2号梯9层门锁信号" := "input"."2号梯9楼层门锁信号";
   "2号梯10层门锁信号" := "input"."2号梯10楼层门锁信号";
END_REGION

REGION Network 11: 3号梯门锁信号
